text := '***';
TOF_Core.Strings.TrimChar(stringToTrim := text, trimChar := '*');
Assert.ThatBool(
	actual := text = '',
	message := "Trimming all matching characters must make the result empty"
).IsTrue();
END_METHOD

//! <summary>Borrows the concrete class name. Callers must not modify it.</summary>
{attribute 'monitoring' := 'call'}
PROPERTY ClassName : REFERENCE TO STRING
GET
ClassName REF= _ClassName;
END_GET
END_PROPERTY

//! <summary>Borrows the compiler-initialized namespace name. Callers must not modify it.</summary>
{attribute 'monitoring' := 'call'}
PROPERTY NamespaceName : REFERENCE TO STRING
GET
NamespaceName REF= CurrentNamespace.Name;
END_GET
END_PROPERTY

//! <summary>Reports the concrete instance size in bytes.</summary>
{attribute 'monitoring' := 'call'}
PROPERTY SelfSize : ULINT
GET
SelfSize := XSIZEOF(THIS^);
END_GET
END_PROPERTY

END_FUNCTION_BLOCK

// ---- Tests/Strings/String/StringSeparatorBoundsTest.TcPOU
(*
SPDX-FileCopyrightText: c 2026 Oleksandr Tiutyk <trofimich@gmail.com>
SPDX-License-Identifier: MIT
License: https://opensource.org/license/mit
*)

(*!
<summary>Checks separator length boundaries and missing borrowed sources.</summary>
<description>
Uses one task and stays at a stable address while assertions are bound to this instance.
</description>
*)

{attribute 'no_assign'}
{attribute 'no_explicit_call' := 'do not call this function block directly'}
FUNCTION_BLOCK StringSeparatorBoundsTest EXTENDS TOF_Testing.SingleCycleTest
VAR_STAT
	{attribute 'hide'}
	_ClassName : STRING := __POUNAME();
END_VAR
VAR
	_Source : STRING(82) := 'xaaaaaaaaaaaaaaaaaaaaaaaaaaaaaaaaaaaaaaaaaaaaaaaaaaaaaaaaaaaaaaaaaaaaaaaaaaaaaaaay';
	_Splitter : TOF_Core.StringSplittingEnumerator;
END_VAR

(*!
<summary>Checks separator length boundaries and missing borrowed sources.</summary>
<description>
Owns a persistent cursor and its borrowed source. The separators are bounded ASCII byte sequences.
Reset releases the current fragment before the result is reported.
</description>
*)
METHOD PROTECTED ExecuteTest
VAR
	separator : STRING(256);
	separatorUnits : POINTER TO BYTE;
	separatorLength : UINT;
	lengths : ARRAY [0..4] OF UINT := [0, 80, 81, 255, 256];
	caseLabel : WSTRING(80);
	missingSource : REFERENCE TO STRING;

	exceptionCode : __SYSTEM.ExceptionCode;
	caught : TOF_Core.IException;
	rangeException : TOF_Core.IArgumentOutOfRangeException;
	accepted : BOOL;
	i : DINT;
	j : INT;
END_VAR
// SA0175: Construct bounded ASCII separators of exact byte lengths.
{analysis -175}
separatorUnits := ADR(separator);
{analysis +175}

FOR i := 0 TO UPPER_BOUND(lengths, 1) DO
	separatorLength := lengths[i];
	caseLabel := Tc2_Utilities.WCONCAT(STR1 := "separator length ", STR2 := TO_WSTRING(separatorLength));
	FOR j := 0 TO TO_INT(separatorLength) - 1 DO
		separatorUnits[j] := BYTE#16#61;
	END_FOR

	separatorUnits[separatorLength] := TO_BYTE(TOF_Core.UnsignedInt8.MIN_VALUE);

	accepted := TOF_Core.Strings.TryCreateSplitter(sourceString := _Source, separator := separator, splitter => _Splitter);
	Assert.ThatBool(
		actual := accepted = (separatorLength = 80),
		message := Tc2_Utilities.WCONCAT(STR1 := "TryCreateSplitter at ", STR2 := caseLabel)
	).IsTrue();

	IF accepted THEN
		assertMaximumSplit(scenario := "TryCreateSplitter must use the full accepted separator");
		_Splitter.Reset();
	END_IF

	caught := 0;

	// Capture the expected argument error before inspecting the payload.
	__TRY
		_Splitter := TOF_Core.Strings.CreateSplitter(sourceString := _Source, separator := separator);
	__CATCH(exceptionCode)
		caught := TOF_Core.ExceptionManager.GetLastException(
			exceptionCode := exceptionCode,
			catchPointNamespaceName := NamespaceName,
			catchPointPOUName := __POUNAME(),
			catchPointPosition := __POSITION()
		);
	__ENDTRY

	IF separatorLength = 80 THEN
		Assert.ThatBool(actual := caught = 0, message := "CreateSplitter must accept length 80").IsTrue();

		IF caught = 0 THEN
			assertMaximumSplit(scenario := "CreateSplitter must use the full accepted separator");
			_Splitter.Reset();
		END_IF
	ELSE
		Assert.ThatBool(
			actual := __QUERYINTERFACE(caught, rangeException),
			message := Tc2_Utilities.WCONCAT(STR1 := "Expected ArgumentOutOfRangeException for ", STR2 := caseLabel)
		).IsTrue();
	END_IF
END_FOR

accepted := TOF_Core.Strings.TryCreateSplitter(
	sourceString := missingSource,
	separator := ',',
	splitter => _Splitter
);
Assert.ThatBool(
	actual := accepted,
	message := "TryCreateSplitter must return FALSE for an unbound source"
).IsFalse();
END_METHOD

(*!
<summary>Verifies that all 80 separator units are used when locating the two fragments.</summary>
<param name="scenario">Factory name included in failure messages.</param>
*)
METHOD PRIVATE assertMaximumSplit
VAR_INPUT
	scenario : WSTRING(80);
END_VAR
VAR
	entry : REFERENCE TO STRING;
	advanced : BOOL;
END_VAR
advanced := _Splitter.MoveNext();
entry REF= _Splitter.CurrentEntry;
Assert.ThatBool(
	actual := advanced AND_THEN __ISVALIDREF(entry) AND_THEN entry = 'x',
	message := scenario
).IsTrue();

advanced := _Splitter.MoveNext();
entry REF= _Splitter.CurrentEntry;
Assert.ThatBool(
	actual := advanced AND_THEN __ISVALIDREF(entry) AND_THEN entry = 'y',
	message := scenario
).IsTrue();

advanced := _Splitter.MoveNext();
Assert.ThatBool(actual := advanced, message := scenario).IsFalse();
END_METHOD

(*!
<summary>Resets the splitter and releases any active fragment before reporting.</summary>
<description>
Safe after partial initialization and after explicit cleanup in the scenario.
</description>
*)
METHOD PROTECTED AfterTest
_Splitter.Reset();
END_METHOD

//! <summary>Borrows the concrete class name. Callers must not modify it.</summary>
{attribute 'monitoring' := 'call'}
PROPERTY ClassName : REFERENCE TO STRING
GET
ClassName REF= _ClassName;
END_GET
END_PROPERTY

//! <summary>Borrows the compiler-initialized namespace name. Callers must not modify it.</summary>
{attribute 'monitoring' := 'call'}
PROPERTY NamespaceName : REFERENCE TO STRING
GET
NamespaceName REF= CurrentNamespace.Name;
END_GET
END_PROPERTY

//! <summary>Reports the concrete instance size in bytes.</summary>
{attribute 'monitoring' := 'call'}
PROPERTY SelfSize : ULINT
GET
SelfSize := XSIZEOF(THIS^);
END_GET
END_PROPERTY

END_FUNCTION_BLOCK

// ---- Tests/Strings/WideString/WideStringsTestGroup.TcPOU
(*
SPDX-FileCopyrightText: c 2026 Oleksandr Tiutyk <trofimich@gmail.com>
SPDX-License-Identifier: MIT
License: https://opensource.org/license/mit
*)

(*!
<summary>Groups wide-string formatting, editing, search and splitter contracts.</summary>
<description>
Owns the independent child instances and their fixed registration array. Use from one PLC task at a stable address.
</description>
*)

{attribute 'no_assign'}
{attribute 'no_explicit_call' := 'do not call this function block directly'}
FUNCTION_BLOCK WideStringsTestGroup EXTENDS TOF_Testing.TestGroup<11>
VAR_STAT
	{attribute 'hide'}
	_ClassName : STRING := __POUNAME();
END_VAR
VAR
	_AnyToStringFit255 : WideStringFitFormattingTest(name := "AnyToStringFit255", parent := THIS^);
	_Append : WideStringAppendTest(name := "Append", parent := THIS^);
	_AppendFit : WideStringAppendFitTest(name := "AppendFit", parent := THIS^);
	_ConcatFit255 : WideStringConcatFitTest(name := "ConcatFit255", parent := THIS^);
	_Contains : WideStringContainsTest(name := "Contains", parent := THIS^);
	_Join : WideStringJoinTest(name := "Join", parent := THIS^);
	_ReplaceInSource : WideStringReplacementTest(name := "ReplaceInSource", parent := THIS^);
	_Split : WideStringSplitTest(name := "Split", parent := THIS^);
	_Trim : WideStringTrimTest(name := "Trim", parent := THIS^);
	_SplitterSeparatorBounds : WideStringSeparatorBoundsTest(name := "SplitterSeparatorBounds", parent := THIS^);
	_AnyToStringFitLongInputs : WideStringLongFitFormattingTest(name := "AnyToStringFitLongInputs", parent := THIS^);

	_Children : ARRAY [0.._ChildCount - 1] OF TOF_Testing.ITestElement :=
	[
		_AnyToStringFit255,
		_Append,
		_AppendFit,
		_ConcatFit255,
		_Contains,
		_Join,
		_ReplaceInSource,
		_Split,
		_Trim,
		_SplitterSeparatorBounds,
		_AnyToStringFitLongInputs
	];
END_VAR

//! <summary>Borrows the fixed child array. Callers must not modify it.</summary>
{attribute 'monitoring' := 'call'}
PROPERTY Children : REFERENCE TO ARRAY [0.._ChildCount - 1] OF TOF_Testing.ITestElement
GET
Children REF= _Children;
END_GET
END_PROPERTY

//! <summary>Borrows the concrete class name. Callers must not modify it.</summary>
{attribute 'monitoring' := 'call'}
PROPERTY ClassName : REFERENCE TO STRING
GET
ClassName REF= _ClassName;
END_GET
END_PROPERTY

//! <summary>Borrows the compiler-initialized namespace name. Callers must not modify it.</summary>
{attribute 'monitoring' := 'call'}
PROPERTY NamespaceName : REFERENCE TO STRING
GET
NamespaceName REF= CurrentNamespace.Name;
END_GET
END_PROPERTY

//! <summary>Reports the concrete instance size in bytes.</summary>
{attribute 'monitoring' := 'call'}
PROPERTY SelfSize : ULINT
GET
SelfSize := XSIZEOF(THIS^);
END_GET
END_PROPERTY

END_FUNCTION_BLOCK

// ---- Tests/Strings/WideString/WideStringFitFormattingTest.TcPOU
(*
SPDX-FileCopyrightText: c 2026 Oleksandr Tiutyk <trofimich@gmail.com>
SPDX-License-Identifier: MIT
License: https://opensource.org/license/mit
*)

(*!
<summary>Checks scalar and short text formatting through the fitted ANY API.</summary>
<description>
Uses one task and stays at a stable address while assertions are bound to this instance.
</description>
*)

{attribute 'no_assign'}
{attribute 'no_explicit_call' := 'do not call this function block directly'}
FUNCTION_BLOCK WideStringFitFormattingTest EXTENDS TOF_Testing.SingleCycleTest
VAR_STAT
	{attribute 'hide'}
	_ClassName : STRING := __POUNAME();
END_VAR

(*!
<summary>Checks scalar and short text formatting through the fitted ANY API.</summary>
*)
METHOD PROTECTED ExecuteTest
VAR
	formatted : WSTRING(255);
	enabled : BOOL := TRUE;
	number : DINT := 12345;
	narrowText : STRING(50) := 'Sample string';
	wideText : WSTRING(50) := "Sample wide string";
END_VAR
formatted := TOF_Core.WideStrings.AnyToStringFit255(value := enabled);
Assert.ThatBool(
	actual := formatted = "TRUE",
	message := "AnyToStringFit255 must format BOOL"
).IsTrue();

formatted := TOF_Core.WideStrings.AnyToStringFit255(value := number);
Assert.ThatBool(
	actual := formatted = "12345",
	message := "AnyToStringFit255 must format DINT"
).IsTrue();

formatted := TOF_Core.WideStrings.AnyToStringFit255(value := narrowText);
Assert.ThatBool(
	actual := formatted = "Sample string",
	message := "AnyToStringFit255 must convert short STRING to WSTRING"
).IsTrue();

formatted := TOF_Core.WideStrings.AnyToStringFit255(value := wideText);
Assert.ThatBool(
	actual := formatted = "Sample wide string",
	message := "AnyToStringFit255 must pass short WSTRING as-is"
).IsTrue();
END_METHOD

//! <summary>Borrows the concrete class name. Callers must not modify it.</summary>
{attribute 'monitoring' := 'call'}
PROPERTY ClassName : REFERENCE TO STRING
GET
ClassName REF= _ClassName;
END_GET
END_PROPERTY

//! <summary>Borrows the compiler-initialized namespace name. Callers must not modify it.</summary>
{attribute 'monitoring' := 'call'}
PROPERTY NamespaceName : REFERENCE TO STRING
GET
NamespaceName REF= CurrentNamespace.Name;
END_GET
END_PROPERTY

//! <summary>Reports the concrete instance size in bytes.</summary>
{attribute 'monitoring' := 'call'}
PROPERTY SelfSize : ULINT
GET
SelfSize := XSIZEOF(THIS^);
END_GET
END_PROPERTY

END_FUNCTION_BLOCK

// ---- Tests/Strings/WideString/WideStringAppendTest.TcPOU
(*
SPDX-FileCopyrightText: c 2026 Oleksandr Tiutyk <trofimich@gmail.com>
SPDX-License-Identifier: MIT
License: https://opensource.org/license/mit
*)

(*!
<summary>Checks strict and Try appends, including empty fragments and capacity failure.</summary>
<description>
Uses one task and stays at a stable address while assertions are bound to this instance.
</description>
*)

{attribute 'no_assign'}
{attribute 'no_explicit_call' := 'do not call this function block directly'}
FUNCTION_BLOCK WideStringAppendTest EXTENDS TOF_Testing.SingleCycleTest
VAR_STAT
	{attribute 'hide'}
	_ClassName : STRING := __POUNAME();
END_VAR

(*!
<summary>Checks strict and Try appends, including empty fragments and capacity failure.</summary>
<description>
Both widths use small buffers to exercise the exact capacity and a failing subsequent append.
</description>
*)
METHOD PROTECTED ExecuteTest
VAR
	target : WSTRING(8);
	accepted : BOOL;
END_VAR
target := "ab";
TOF_Core.WideStrings.Append255(target, "cd", "", "efgh");
Assert.ThatBool(
	actual := target = "abcdefgh",
	message := "Append255 must skip an empty fragment and fill the target exactly"
).IsTrue();

target := "ab";
accepted := TOF_Core.WideStrings.TryAppend255(
	targetString := target,
	sourceString1 := "cd",
	sourceString2 := "",
	sourceString3 := "efgh"
);
Assert.ThatBool(
	actual := accepted AND_THEN target = "abcdefgh",
	message := "TryAppend255 must accept an exact fit"
).IsTrue();

target := "ab";
accepted := TOF_Core.WideStrings.TryAppend255(
	targetString := target,
	sourceString1 := "cd",
	sourceString2 := "ABCDE",
	sourceString3 := "!"
);
Assert.ThatBool(
	actual := accepted,
	message := "TryAppend255 must report capacity failure"
).IsFalse();
Assert.ThatBool(
	actual := Tc2_Standard.WLEFT(STR := target, SIZE := 4) = "abcd",
	message := "TryAppend255 must preserve the successfully appended prefix"
).IsTrue();

target := "ab";
TOF_Core.WideStrings.Append(targetString := target, sourceString := "cd");
TOF_Core.WideStrings.Append(targetString := target, sourceString := "");
TOF_Core.WideStrings.Append(targetString := target, sourceString := "efgh");
Assert.ThatBool(
	actual := target = "abcdefgh",
	message := "Append must preserve the target on empty input and accept the exact fit"
).IsTrue();

target := "abcdef";
accepted := TOF_Core.WideStrings.TryAppend(targetString := target, sourceString := "gh");
Assert.ThatBool(
	actual := accepted AND_THEN target = "abcdefgh",
	message := "TryAppend must accept an exact fit"
).IsTrue();

accepted := TOF_Core.WideStrings.TryAppend(targetString := target, sourceString := "i");
Assert.ThatBool(
	actual := accepted,
	message := "TryAppend must reject another character in a full target"
).IsFalse();
Assert.ThatBool(
	actual := target = "abcdefgh",
	message := "TryAppend must preserve the full target when one more character does not fit"
).IsTrue();
END_METHOD

//! <summary>Borrows the concrete class name. Callers must not modify it.</summary>
{attribute 'monitoring' := 'call'}
PROPERTY ClassName : REFERENCE TO STRING
GET
ClassName REF= _ClassName;
END_GET
END_PROPERTY

//! <summary>Borrows the compiler-initialized namespace name. Callers must not modify it.</summary>
{attribute 'monitoring' := 'call'}
PROPERTY NamespaceName : REFERENCE TO STRING
GET
NamespaceName REF= CurrentNamespace.Name;
END_GET
END_PROPERTY

//! <summary>Reports the concrete instance size in bytes.</summary>
{attribute 'monitoring' := 'call'}
PROPERTY SelfSize : ULINT
GET
SelfSize := XSIZEOF(THIS^);
END_GET
END_PROPERTY

END_FUNCTION_BLOCK

// ---- Tests/Strings/WideString/WideStringAppendFitTest.TcPOU
(*
SPDX-FileCopyrightText: c 2026 Oleksandr Tiutyk <trofimich@gmail.com>
SPDX-License-Identifier: MIT
License: https://opensource.org/license/mit
*)

(*!
<summary>Checks fitted appends at exact capacity and on truncation.</summary>
<description>
Uses one task and stays at a stable address while assertions are bound to this instance.
</description>
*)

{attribute 'no_assign'}
{attribute 'no_explicit_call' := 'do not call this function block directly'}
FUNCTION_BLOCK WideStringAppendFitTest EXTENDS TOF_Testing.SingleCycleTest
VAR_STAT
	{attribute 'hide'}
	_ClassName : STRING := __POUNAME();
END_VAR

(*!
<summary>Checks fitted appends at exact capacity and on truncation.</summary>
*)
METHOD PROTECTED ExecuteTest
VAR
	oneCharacter : WSTRING(1);
	twoCharacters : WSTRING(2);
	target : WSTRING(10);
	longFragment : WSTRING(30) := "01234567890123456789";
	accepted : BOOL;
END_VAR
// Fits within capacity
target := "12345";
TOF_Core.WideStrings.AppendFit(targetString := target, sourceString := "67");
Assert.ThatBool(
	actual := target = "1234567",
	message := "AppendFit must append normally when it fits"
).IsTrue();

// Exact fit: fills capacity without ellipsis
target := "12345";
TOF_Core.WideStrings.AppendFit(targetString := target, sourceString := "67890");
Assert.ThatBool(
	actual := target = "1234567890",
	message := "AppendFit must fit exactly without ellipsis"
).IsTrue();

// Overflow by one code unit uses U+2026.
target := "12345";
TOF_Core.WideStrings.AppendFit(targetString := target, sourceString := "678901");
Assert.ThatBool(
	actual := target = "123456789$2026",
	message := "AppendFit must truncate and append ellipsis on 1 char overflow"
).IsTrue();

// A larger overflow still uses one U+2026 code unit.
target := "12345";
TOF_Core.WideStrings.AppendFit(targetString := target, sourceString := longFragment);
Assert.ThatBool(
	actual := target = "123450123$2026",
	message := "AppendFit must truncate and append ellipsis on large overflow"
).IsTrue();

// Empty source: target remains unchanged
target := "12345";
TOF_Core.WideStrings.AppendFit(targetString := target, sourceString := "");
Assert.ThatBool(
	actual := target = "12345",
	message := "AppendFit must leave target unchanged for empty source"
).IsTrue();

// Appending to empty target
target := "";
TOF_Core.WideStrings.AppendFit(targetString := target, sourceString := longFragment);
Assert.ThatBool(
	actual := target = "012345678$2026",
	message := "AppendFit to empty target must truncate and append ellipsis"
).IsTrue();

// TryAppendFit normal fit
target := "123";
accepted := TOF_Core.WideStrings.TryAppendFit(targetString := target, sourceString := "45");
Assert.ThatBool(
	actual := accepted,
	message := "TryAppendFit must return TRUE on normal fit"
).IsTrue();
Assert.ThatBool(
	actual := target = "12345",
	message := "TryAppendFit must append text"
).IsTrue();

// TryAppendFit overflow
target := "12345";
accepted := TOF_Core.WideStrings.TryAppendFit(targetString := target, sourceString := longFragment);
Assert.ThatBool(
	actual := accepted,
	message := "TryAppendFit must return TRUE on overflow"
).IsTrue();
Assert.ThatBool(
	actual := target = "123450123$2026",
	message := "TryAppendFit must truncate and append ellipsis"
).IsTrue();

// AppendFit255 multiple arguments and literals
target := "12";
TOF_Core.WideStrings.AppendFit255(target, "3", "4", "5");
Assert.ThatBool(
	actual := target = "12345",
	message := "AppendFit255 must append multiple fragments"
).IsTrue();

// AppendFit255 overflow truncation
target := "12";
TOF_Core.WideStrings.AppendFit255(target, "345", "678", "9012");
Assert.ThatBool(
	actual := target = "123456789$2026",
	message := "AppendFit255 must truncate and append ellipsis on overflow"
).IsTrue();

// TryAppendFit255 normal fit
target := "12";
accepted := TOF_Core.WideStrings.TryAppendFit255(
	targetString := target,
	sourceString1 := "3",
	sourceString2 := "4",
	sourceString3 := "5"
);
Assert.ThatBool(
	actual := accepted,
	message := "TryAppendFit255 must return TRUE on normal fit"
).IsTrue();
Assert.ThatBool(
	actual := target = "12345",
	message := "TryAppendFit255 must append multiple fragments"
).IsTrue();

// TryAppendFit255 overflow
target := "12";
accepted := TOF_Core.WideStrings.TryAppendFit255(
	targetString := target,
	sourceString1 := "345",
	sourceString2 := "678",
	sourceString3 := "9012"
);
Assert.ThatBool(
	actual := accepted,
	message := "TryAppendFit255 must return TRUE on overflow"
).IsTrue();
Assert.ThatBool(
	actual := target = "123456789$2026",
	message := "TryAppendFit255 must truncate and append ellipsis on overflow"
).IsTrue();

accepted := TOF_Core.WideStrings.TryAppendFit(targetString := oneCharacter, sourceString := longFragment);
Assert.ThatBool(
	actual := accepted,
	message := "Truncation must succeed in a one-character buffer"
).IsTrue();
Assert.ThatBool(
	actual := oneCharacter = "$2026",
	message := "One-character truncation marker"
).IsTrue();

accepted := TOF_Core.WideStrings.TryAppendFit255(targetString := twoCharacters, sourceString1 := longFragment);
Assert.ThatBool(
	actual := accepted,
	message := "Truncation must succeed in a two-character buffer"
).IsTrue();
Assert.ThatBool(
	actual := twoCharacters = "0$2026",
	message := "Two-character truncation marker"
).IsTrue();
END_METHOD

//! <summary>Borrows the concrete class name. Callers must not modify it.</summary>
{attribute 'monitoring' := 'call'}
PROPERTY ClassName : REFERENCE TO STRING
GET
ClassName REF= _ClassName;
END_GET
END_PROPERTY

//! <summary>Borrows the compiler-initialized namespace name. Callers must not modify it.</summary>
{attribute 'monitoring' := 'call'}
PROPERTY NamespaceName : REFERENCE TO STRING
GET
NamespaceName REF= CurrentNamespace.Name;
END_GET
END_PROPERTY

//! <summary>Reports the concrete instance size in bytes.</summary>
{attribute 'monitoring' := 'call'}
PROPERTY SelfSize : ULINT
GET
SelfSize := XSIZEOF(THIS^);
END_GET
END_PROPERTY

END_FUNCTION_BLOCK

// ---- Tests/Strings/WideString/WideStringConcatFitTest.TcPOU
(*
SPDX-FileCopyrightText: c 2026 Oleksandr Tiutyk <trofimich@gmail.com>
SPDX-License-Identifier: MIT
License: https://opensource.org/license/mit
*)

(*!
<summary>Checks fitted concatenation, including the 255-character boundary.</summary>
<description>
Uses one task and stays at a stable address while assertions are bound to this instance.
</description>
*)

{attribute 'no_assign'}
{attribute 'no_explicit_call' := 'do not call this function block directly'}
FUNCTION_BLOCK WideStringConcatFitTest EXTENDS TOF_Testing.SingleCycleTest
VAR_STAT
	{attribute 'hide'}
	_ClassName : STRING := __POUNAME();
END_VAR

(*!
<summary>Checks fitted concatenation, including the 255-character boundary.</summary>
<description>
Distinct fragments reveal the first discarded character and any changes in fragment order.
</description>
*)
METHOD PROTECTED ExecuteTest
VAR
	text : WSTRING(255);
	first : WSTRING(100) := "aaaaaaaaaaaaaaaaaaaaaaaaaaaaaaaaaaaaaaaaaaaaaaaaaaaaaaaaaaaaaaaaaaaaaaaaaaaaaaaaaaaaaaaaaaaaaaaaaaaa";
	second : WSTRING(100) := "bbbbbbbbbbbbbbbbbbbbbbbbbbbbbbbbbbbbbbbbbbbbbbbbbbbbbbbbbbbbbbbbbbbbbbbbbbbbbbbbbbbbbbbbbbbbbbbbbbbb";
	third : WSTRING(100) := "cccccccccccccccccccccccccccccccccccccccccccccccccccccccccccccccccccccccccccccccccccccccccccccccccccc";
	expectedPrefix : WSTRING(255);
END_VAR
text := TOF_Core.WideStrings.ConcatFit255("Hello, ", "World!");
Assert.ThatBool(
	actual := text = "Hello, World!",
	message := "ConcatFit255 must preserve an ordinary fit"
).IsTrue();

text := TOF_Core.WideStrings.ConcatFit255("Part1", "", "Part2", "", "Part3");
Assert.ThatBool(
	actual := text = "Part1Part2Part3",
	message := "ConcatFit255 must skip empty fragments without stopping"
).IsTrue();

text := TOF_Core.WideStrings.ConcatFit255(first, second, third);
Assert.ThatInt(
	actual := Tc2_Standard.WLEN(STR := text),
	message := "ConcatFit255 must fill the 255-character result"
).ToBe(expected := 255);
expectedPrefix := Tc2_Standard.WCONCAT(STR1 := first, STR2 := second);
expectedPrefix := Tc2_Standard.WCONCAT(
	STR1 := expectedPrefix,
	STR2 := Tc2_Standard.WLEFT(STR := third, SIZE := 54)
);
Assert.ThatBool(
	actual := Tc2_Standard.WLEFT(STR := text, SIZE := 254) = expectedPrefix,
	message := "Truncation must preserve the prefix across all three fragments"
).IsTrue();
Assert.ThatBool(
	actual := Tc2_Standard.WRIGHT(STR := text, SIZE := 1) = "$2026",
	message := "Truncation must use the exact encoding-specific ellipsis"
).IsTrue();
END_METHOD

//! <summary>Borrows the concrete class name. Callers must not modify it.</summary>
{attribute 'monitoring' := 'call'}
PROPERTY ClassName : REFERENCE TO STRING
GET
ClassName REF= _ClassName;
END_GET
END_PROPERTY

//! <summary>Borrows the compiler-initialized namespace name. Callers must not modify it.</summary>
{attribute 'monitoring' := 'call'}
PROPERTY NamespaceName : REFERENCE TO STRING
GET
NamespaceName REF= CurrentNamespace.Name;
END_GET
END_PROPERTY

//! <summary>Reports the concrete instance size in bytes.</summary>
{attribute 'monitoring' := 'call'}
PROPERTY SelfSize : ULINT
GET
SelfSize := XSIZEOF(THIS^);
END_GET
END_PROPERTY

END_FUNCTION_BLOCK

// ---- Tests/Strings/WideString/WideStringContainsTest.TcPOU
(*
SPDX-FileCopyrightText: c 2026 Oleksandr Tiutyk <trofimich@gmail.com>
SPDX-License-Identifier: MIT
License: https://opensource.org/license/mit
*)

(*!
<summary>Checks exact, case-sensitive substring matching and empty inputs.</summary>
<description>
Uses one task and stays at a stable address while assertions are bound to this instance.
</description>
*)

{attribute 'no_assign'}
{attribute 'no_explicit_call' := 'do not call this function block directly'}
FUNCTION_BLOCK WideStringContainsTest EXTENDS TOF_Testing.SingleCycleTest
VAR_STAT
	{attribute 'hide'}
	_ClassName : STRING := __POUNAME();
END_VAR

(*!
<summary>Checks exact, case-sensitive substring matching and empty inputs.</summary>
*)
METHOD PROTECTED ExecuteTest
VAR
	containsResult : BOOL;
END_VAR
containsResult := TOF_Core.WideStrings.Contains(stringToSearchIn := "Hello, world!", stringToFind := "Hello");
Assert.ThatBool(
	actual := containsResult,
	message := "Contains must return TRUE for prefix substring"
).IsTrue();

containsResult := TOF_Core.WideStrings.Contains(stringToSearchIn := "Hello, world!", stringToFind := "world");
Assert.ThatBool(
	actual := containsResult,
	message := "Contains must return TRUE for middle substring"
).IsTrue();

containsResult := TOF_Core.WideStrings.Contains(stringToSearchIn := "Hello, world!", stringToFind := "!");
Assert.ThatBool(
	actual := containsResult,
	message := "Contains must return TRUE for suffix substring"
).IsTrue();

containsResult := TOF_Core.WideStrings.Contains(stringToSearchIn := "Hello, world!", stringToFind := "Hello, world!");
Assert.ThatBool(
	actual := containsResult,
	message := "Contains must return TRUE for identical string"
).IsTrue();

containsResult := TOF_Core.WideStrings.Contains(stringToSearchIn := "Hello, world!", stringToFind := "");
Assert.ThatBool(
	actual := containsResult,
	message := "Contains must return TRUE for empty substring in non-empty string"
).IsTrue();

containsResult := TOF_Core.WideStrings.Contains(stringToSearchIn := "", stringToFind := "");
Assert.ThatBool(
	actual := containsResult,
	message := "Contains must return TRUE for empty substring in empty string"
).IsTrue();

containsResult := TOF_Core.WideStrings.Contains(stringToSearchIn := "", stringToFind := "a");
Assert.ThatBool(
	actual := containsResult,
	message := "Contains must return FALSE for non-empty substring in empty string"
).IsFalse();

containsResult := TOF_Core.WideStrings.Contains(stringToSearchIn := "Hello, world!", stringToFind := "xyz");
Assert.ThatBool(
	actual := containsResult,
	message := "Contains must return FALSE when substring is absent"
).IsFalse();

containsResult := TOF_Core.WideStrings.Contains(stringToSearchIn := "Hello, world!", stringToFind := "hello");
Assert.ThatBool(
	actual := containsResult,
	message := "Contains must be case-sensitive"
).IsFalse();

containsResult := TOF_Core.WideStrings.Contains(stringToSearchIn := "abc", stringToFind := "abcdef");
Assert.ThatBool(
	actual := containsResult,
	message := "Contains must return FALSE when substring is longer than source"
).IsFalse();

containsResult := TOF_Core.WideStrings.Contains(stringToSearchIn := "aaab", stringToFind := "aab");
Assert.ThatBool(
	actual := containsResult,
	message := "Contains must restart after a partially matching prefix"
).IsTrue();
END_METHOD

//! <summary>Borrows the concrete class name. Callers must not modify it.</summary>
{attribute 'monitoring' := 'call'}
PROPERTY ClassName : REFERENCE TO STRING
GET
ClassName REF= _ClassName;
END_GET
END_PROPERTY

//! <summary>Borrows the compiler-initialized namespace name. Callers must not modify it.</summary>
{attribute 'monitoring' := 'call'}
PROPERTY NamespaceName : REFERENCE TO STRING
GET
NamespaceName REF= CurrentNamespace.Name;
END_GET
END_PROPERTY

//! <summary>Reports the concrete instance size in bytes.</summary>
{attribute 'monitoring' := 'call'}
PROPERTY SelfSize : ULINT
GET
SelfSize := XSIZEOF(THIS^);
END_GET
END_PROPERTY

END_FUNCTION_BLOCK

// ---- Tests/Strings/WideString/WideStringJoinTest.TcPOU
(*
SPDX-FileCopyrightText: c 2026 Oleksandr Tiutyk <trofimich@gmail.com>
SPDX-License-Identifier: MIT
License: https://opensource.org/license/mit
*)

(*!
<summary>Checks full and windowed joining and cursor reuse after insufficient capacity.</summary>
<description>
Uses one task and stays at a stable address while assertions are bound to this instance.
</description>
*)

{attribute 'no_assign'}
{attribute 'no_explicit_call' := 'do not call this function block directly'}
FUNCTION_BLOCK WideStringJoinTest EXTENDS TOF_Testing.SingleCycleTest
VAR_STAT
	{attribute 'hide'}
	_ClassName : STRING := __POUNAME();
END_VAR
VAR
	_Source : WSTRING := "123 , , 456, 789 ,0";
	_Splitter : TOF_Core.WideStringSplittingEnumerator;
END_VAR

(*!
<summary>Checks full and windowed joining and cursor reuse after insufficient capacity.</summary>
<description>
Owns a persistent cursor and its borrowed source. Reset releases the current fragment before the result is reported.
</description>
*)
METHOD PROTECTED ExecuteTest
VAR
	separator : WSTRING := ",";
	joined : WSTRING := "old target";
	shortTarget : WSTRING(2);
	accepted : BOOL;
END_VAR
_Splitter := TOF_Core.WideStrings.CreateSplitter(sourceString := _Source, separator := separator);
TOF_Core.WideStrings.Join(targetString := joined, separator := separator, sourceEnumerator := _Splitter);
Assert.ThatBool(
	actual := joined = _Source,
	message := "Unrestricted Join must reconstruct all fragments including their whitespace"
).IsTrue();

_Splitter.Reset();
_Splitter := TOF_Core.WideStrings.CreateSplitter(
	sourceString := _Source,
	separator := separator,
	maxCount := 3,
	trimEntries := TRUE,
	removeEmptyEntries := TRUE
);
TOF_Core.WideStrings.Join(
	targetString := joined,
	separator := separator,
	sourceEnumerator := _Splitter,
	startIndex := 1,
	count := 2
);
Assert.ThatBool(
	actual := joined = "456,789",
	message := "The requested window must contain fragments 1 and 2"
).IsTrue();

_Splitter.Reset();
accepted := TOF_Core.WideStrings.TryJoin(targetString := shortTarget, separator := separator, sourceEnumerator := _Splitter);
Assert.ThatBool(
	actual := accepted,
	message := "TryJoin must reject a target too small for the first fragment"
).IsFalse();

_Splitter.Reset();
accepted := TOF_Core.WideStrings.TryJoin(
	targetString := joined,
	separator := separator,
	sourceEnumerator := _Splitter,
	count := 1
);
Assert.ThatBool(
	actual := accepted AND_THEN joined = "123",
	message := "After Reset, TryJoin must restart and replace the old target text"
).IsTrue();
END_METHOD

(*!
<summary>Resets the splitter and releases any active fragment before reporting.</summary>
<description>
Safe after partial initialization and after explicit cleanup in the scenario.
</description>
*)
METHOD PROTECTED AfterTest
_Splitter.Reset();
END_METHOD

//! <summary>Borrows the concrete class name. Callers must not modify it.</summary>
{attribute 'monitoring' := 'call'}
PROPERTY ClassName : REFERENCE TO STRING
GET
ClassName REF= _ClassName;
END_GET
END_PROPERTY

//! <summary>Borrows the compiler-initialized namespace name. Callers must not modify it.</summary>
{attribute 'monitoring' := 'call'}
PROPERTY NamespaceName : REFERENCE TO STRING
GET
NamespaceName REF= CurrentNamespace.Name;
END_GET
END_PROPERTY

//! <summary>Reports the concrete instance size in bytes.</summary>
{attribute 'monitoring' := 'call'}
PROPERTY SelfSize : ULINT
GET
SelfSize := XSIZEOF(THIS^);
END_GET
END_PROPERTY

END_FUNCTION_BLOCK

// ---- Tests/Strings/WideString/WideStringReplacementTest.TcPOU
(*
SPDX-FileCopyrightText: c 2026 Oleksandr Tiutyk <trofimich@gmail.com>
SPDX-License-Identifier: MIT
License: https://opensource.org/license/mit
*)

(*!
<summary>Checks in-place replacements, counts, limits and partial capacity failure.</summary>
<description>
Uses one task and stays at a stable address while assertions are bound to this instance.
</description>
*)

{attribute 'no_assign'}
{attribute 'no_explicit_call' := 'do not call this function block directly'}
FUNCTION_BLOCK WideStringReplacementTest EXTENDS TOF_Testing.SingleCycleTest
VAR_STAT
	{attribute 'hide'}
	_ClassName : STRING := __POUNAME();
END_VAR

(*!
<summary>Checks in-place replacements, counts, limits and partial capacity failure.</summary>
<description>
Uses caller-owned buffers with known capacities. A failed next replacement must leave earlier matches applied.
</description>
*)
METHOD PROTECTED ExecuteTest
VAR
	text : WSTRING(18);
	
	replacementCount : UINT;
	result : BOOL;
END_VAR
text := "abcd_abcd_abcd";
TOF_Core.WideStrings.ReplaceInSource(
	sourceString := text,
	oldSubstring := "bc",
	newSubstring := "0",
	replacementCount => replacementCount
);
Assert.ThatBool(
	actual := text = "a0d_a0d_a0d",
	message := "Shrink must produce the expected text"
).IsTrue();
Assert.ThatUInt(
	actual := replacementCount,
	message := "Shrink must produce the expected count"
).ToBe(expected := 3);

text := "abcd_abcd_abcd";
TOF_Core.WideStrings.ReplaceInSource(
	sourceString := text,
	oldSubstring := "bc",
	newSubstring := "123",
	replacementCount => replacementCount
);
Assert.ThatBool(
	actual := text = "a123d_a123d_a123d",
	message := "Grow must produce the expected text"
).IsTrue();
Assert.ThatUInt(
	actual := replacementCount,
	message := "Grow must produce the expected count"
).ToBe(expected := 3);

text := "abcd_abcd_abcd";
result := TOF_Core.WideStrings.TryReplaceInSource(
	sourceString := text,
	oldSubstring := "bc",
	newSubstring := "0",
	replacementCount => replacementCount
);
Assert.ThatBool(
	actual := result,
	message := "Try shrink must produce the expected status"
).IsTrue();
Assert.ThatBool(
	actual := text = "a0d_a0d_a0d",
	message := "Try shrink must produce the expected text"
).IsTrue();
Assert.ThatUInt(
	actual := replacementCount,
	message := "Try shrink must produce the expected count"
).ToBe(expected := 3);

text := "abcd_abcd_abcd";
result := TOF_Core.WideStrings.TryReplaceInSource(
	sourceString := text,
	oldSubstring := "bc",
	newSubstring := "123",
	maxReplacements := 1,
	skipReplacements := 1,
	replacementCount => replacementCount
);
Assert.ThatBool(
	actual := result,
	message := "Try skip and limit must produce the expected status"
).IsTrue();
Assert.ThatBool(
	actual := text = "abcd_a123d_abcd",
	message := "Try skip and limit must produce the expected text"
).IsTrue();
Assert.ThatUInt(
	actual := replacementCount,
	message := "Try skip and limit must produce the expected count"
).ToBe(expected := 1);

text := "abcd_abcd_abcd";
result := TOF_Core.WideStrings.TryReplaceInSource(
	sourceString := text,
	oldSubstring := "bc",
	newSubstring := "1234",
	replacementCount => replacementCount
);
Assert.ThatBool(
	actual := result,
	message := "Growth must report failure when the next replacement exceeds capacity"
).IsFalse();
Assert.ThatBool(
	actual := text = "a1234d_a1234d_abcd",
	message := "Capacity failure must preserve both completed replacements"
).IsTrue();
Assert.ThatUInt(
	actual := replacementCount,
	message := "Capacity failure must report both completed replacements"
).ToBe(expected := UINT#2);

text := "abcd_abcd";
result := TOF_Core.WideStrings.TryReplaceInSource(
	sourceString := text,
	oldSubstring := "",
	newSubstring := "ignore",
	replacementCount => replacementCount
);
Assert.ThatBool(
	actual := result AND_THEN text = "abcd_abcd" AND_THEN replacementCount = 0,
	message := "An empty search must succeed without modifying text or reporting replacements"
).IsTrue();

result := TOF_Core.WideStrings.TryReplaceInSource(
	sourceString := text,
	oldSubstring := "bc",
	newSubstring := "",
	replacementCount => replacementCount
);
Assert.ThatBool(
	actual := result AND_THEN text = "ad_ad" AND_THEN replacementCount = 2,
	message := "An empty replacement must delete both matching substrings"
).IsTrue();
END_METHOD

//! <summary>Borrows the concrete class name. Callers must not modify it.</summary>
{attribute 'monitoring' := 'call'}
PROPERTY ClassName : REFERENCE TO STRING
GET
ClassName REF= _ClassName;
END_GET
END_PROPERTY

//! <summary>Borrows the compiler-initialized namespace name. Callers must not modify it.</summary>
{attribute 'monitoring' := 'call'}
PROPERTY NamespaceName : REFERENCE TO STRING
GET
NamespaceName REF= CurrentNamespace.Name;
END_GET
END_PROPERTY

//! <summary>Reports the concrete instance size in bytes.</summary>
{attribute 'monitoring' := 'call'}
PROPERTY SelfSize : ULINT
GET
SelfSize := XSIZEOF(THIS^);
END_GET
END_PROPERTY

END_FUNCTION_BLOCK

// ---- Tests/Strings/WideString/WideStringSplitTest.TcPOU
(*
SPDX-FileCopyrightText: c 2026 Oleksandr Tiutyk <trofimich@gmail.com>
SPDX-License-Identifier: MIT
License: https://opensource.org/license/mit
*)

(*!
<summary>Checks split fragments, end-of-iteration behavior and cursor restart.</summary>
<description>
Uses one task and stays at a stable address while assertions are bound to this instance.
</description>
*)

{attribute 'no_assign'}
{attribute 'no_explicit_call' := 'do not call this function block directly'}
FUNCTION_BLOCK WideStringSplitTest EXTENDS TOF_Testing.SingleCycleTest
VAR_STAT
	{attribute 'hide'}
	_ClassName : STRING := __POUNAME();
END_VAR
VAR
	_Source : WSTRING := "123 , 456, 789 ,,0,";
	_Splitter : TOF_Core.WideStringSplittingEnumerator;
END_VAR

(*!
<summary>Checks split fragments, end-of-iteration behavior and cursor restart.</summary>
<description>
Owns a persistent cursor and its borrowed source. Reset releases the current fragment before the result is reported.
</description>
*)
METHOD PROTECTED ExecuteTest
VAR
	separator : WSTRING := ",";
	allFragments : ARRAY [0..5] OF WSTRING := ["123 ", " 456", " 789 ", "", "0", ""];
	selectedFragments : ARRAY [0..2] OF WSTRING := ["123", "456", "789"];
	entry : REFERENCE TO WSTRING;
	advanced : BOOL;
END_VAR
_Splitter := TOF_Core.WideStrings.CreateSplitter(sourceString := _Source, separator := separator);
assertFragments(expected := allFragments, scenario := "Unrestricted split");

_Splitter.Reset();
_Splitter := TOF_Core.WideStrings.CreateSplitter(
	sourceString := _Source,
	separator := separator,
	maxCount := 3,
	trimEntries := TRUE,
	removeEmptyEntries := TRUE
);
assertFragments(expected := selectedFragments, scenario := "Trimmed split limited to three");

_Splitter.Reset();
entry REF= _Splitter.CurrentEntry;
Assert.ThatBool(
	actual := __ISVALIDREF(entry),
	message := "Reset must leave CurrentEntry invalid until the next successful move"
).IsFalse();

advanced := _Splitter.MoveNext();
entry REF= _Splitter.CurrentEntry;
Assert.ThatBool(
	actual := advanced AND_THEN __ISVALIDREF(entry) AND_THEN entry = "123",
	message := "After Reset the first trimmed fragment must be available again"
).IsTrue();
END_METHOD

(*!
<summary>Checks the requested finite sequence and detects trailing fragments or a stale current reference.</summary>
<param name="expected">Expected fragments in order.</param>
<param name="scenario">Cursor configuration included in failure messages.</param>
*)
METHOD PRIVATE assertFragments
VAR_IN_OUT CONSTANT
	expected : ARRAY [*] OF WSTRING;
END_VAR
VAR_INPUT
	scenario : WSTRING(80);
END_VAR
VAR
	entry : REFERENCE TO WSTRING;
	i : DINT;
	advanced : BOOL;
	fragmentLabel : WSTRING(255);
END_VAR
FOR i := LOWER_BOUND(expected, 1) TO UPPER_BOUND(expected, 1) DO
	fragmentLabel := Tc2_Utilities.WCONCAT(STR1 := scenario, STR2 := " fragment ");
	fragmentLabel := Tc2_Utilities.WCONCAT(STR1 := fragmentLabel, STR2 := TO_WSTRING(i));
	advanced := _Splitter.MoveNext();
	Assert.ThatBool(actual := advanced, message := fragmentLabel).IsTrue();

	IF NOT advanced THEN
		RETURN;
	END_IF

	entry REF= _Splitter.CurrentEntry;
	Assert.ThatBool(actual := __ISVALIDREF(entry) AND_THEN entry = expected[i], message := fragmentLabel).IsTrue();
END_FOR

advanced := _Splitter.MoveNext();
Assert.ThatBool(
	actual := advanced,
	message := Tc2_Utilities.WCONCAT(STR1 := "Unexpected extra fragment in ", STR2 := scenario)
).IsFalse();

IF advanced THEN
	RETURN;
END_IF

entry REF= _Splitter.CurrentEntry;
Assert.ThatBool(actual := __ISVALIDREF(entry), message := "End of iteration must invalidate CurrentEntry").IsFalse();
advanced := _Splitter.MoveNext();
Assert.ThatBool(actual := advanced, message := "An exhausted splitter must stay exhausted").IsFalse();
END_METHOD

(*!
<summary>Resets the splitter and releases any active fragment before reporting.</summary>
<description>
Safe after partial initialization and after explicit cleanup in the scenario.
</description>
*)
METHOD PROTECTED AfterTest
_Splitter.Reset();
END_METHOD

//! <summary>Borrows the concrete class name. Callers must not modify it.</summary>
{attribute 'monitoring' := 'call'}
PROPERTY ClassName : REFERENCE TO STRING
GET
ClassName REF= _ClassName;
END_GET
END_PROPERTY

//! <summary>Borrows the compiler-initialized namespace name. Callers must not modify it.</summary>
{attribute 'monitoring' := 'call'}
PROPERTY NamespaceName : REFERENCE TO STRING
GET
NamespaceName REF= CurrentNamespace.Name;
END_GET
END_PROPERTY

//! <summary>Reports the concrete instance size in bytes.</summary>
{attribute 'monitoring' := 'call'}
PROPERTY SelfSize : ULINT
GET
SelfSize := XSIZEOF(THIS^);
END_GET
END_PROPERTY

END_FUNCTION_BLOCK

// ---- Tests/Strings/WideString/WideStringTrimTest.TcPOU
(*
SPDX-FileCopyrightText: c 2026 Oleksandr Tiutyk <trofimich@gmail.com>
SPDX-License-Identifier: MIT
License: https://opensource.org/license/mit
*)

(*!
<summary>Checks trimming direction, custom characters and complete removal.</summary>
<description>
Uses one task and stays at a stable address while assertions are bound to this instance.
</description>
*)

{attribute 'no_assign'}
{attribute 'no_explicit_call' := 'do not call this function block directly'}
FUNCTION_BLOCK WideStringTrimTest EXTENDS TOF_Testing.SingleCycleTest
VAR_STAT
	{attribute 'hide'}
	_ClassName : STRING := __POUNAME();
END_VAR

(*!
<summary>Checks trimming direction, custom characters and complete removal.</summary>
*)
METHOD PROTECTED ExecuteTest
VAR
	text : WSTRING;
END_VAR
text := "  123   ";
TOF_Core.WideStrings.TrimChar(stringToTrim := text, trimMode := TOF_Core.TRIM_MODE.LEFT_AND_RIGHT);
Assert.ThatBool(
	actual := text = "123",
	message := "TrimChar must apply LEFT_AND_RIGHT exactly"
).IsTrue();

text := "  123   ";
TOF_Core.WideStrings.TrimChar(stringToTrim := text, trimMode := TOF_Core.TRIM_MODE.LEFT);
Assert.ThatBool(
	actual := text = "123   ",
	message := "TrimChar must apply LEFT exactly"
).IsTrue();

text := "  123   ";
TOF_Core.WideStrings.TrimChar(stringToTrim := text, trimMode := TOF_Core.TRIM_MODE.RIGHT);
Assert.ThatBool(
	actual := text = "  123",
	message := "TrimChar must apply RIGHT exactly"
).IsTrue();

text := "**a*b**";
TOF_Core.WideStrings.TrimChar(stringToTrim := text, trimMode := TOF_Core.TRIM_MODE.LEFT_AND_RIGHT, trimChar := "*");
Assert.ThatBool(
	actual := text = "a*b",
	message := "Trimming a custom character must preserve an internal match"
).IsTrue();

text := "***";
TOF_Core.WideStrings.TrimChar(stringToTrim := text, trimChar := "*");
Assert.ThatBool(
	actual := text = "",
	message := "Trimming all matching characters must make the result empty"
).IsTrue();
END_METHOD

//! <summary>Borrows the concrete class name. Callers must not modify it.</summary>
{attribute 'monitoring' := 'call'}
PROPERTY ClassName : REFERENCE TO STRING
GET
ClassName REF= _ClassName;
END_GET
END_PROPERTY

//! <summary>Borrows the compiler-initialized namespace name. Callers must not modify it.</summary>
{attribute 'monitoring' := 'call'}
PROPERTY NamespaceName : REFERENCE TO STRING
GET
NamespaceName REF= CurrentNamespace.Name;
END_GET
END_PROPERTY

//! <summary>Reports the concrete instance size in bytes.</summary>
{attribute 'monitoring' := 'call'}
PROPERTY SelfSize : ULINT
GET
SelfSize := XSIZEOF(THIS^);
END_GET
END_PROPERTY

END_FUNCTION_BLOCK

// ---- Tests/Strings/WideString/WideStringSeparatorBoundsTest.TcPOU
(*
SPDX-FileCopyrightText: c 2026 Oleksandr Tiutyk <trofimich@gmail.com>
SPDX-License-Identifier: MIT
License: https://opensource.org/license/mit
*)

(*!
<summary>Checks separator length boundaries and missing borrowed sources.</summary>
<description>
Uses one task and stays at a stable address while assertions are bound to this instance.
</description>
*)

{attribute 'no_assign'}
{attribute 'no_explicit_call' := 'do not call this function block directly'}
FUNCTION_BLOCK WideStringSeparatorBoundsTest EXTENDS TOF_Testing.SingleCycleTest
VAR_STAT
	{attribute 'hide'}
	_ClassName : STRING := __POUNAME();
END_VAR
VAR
	_Source : WSTRING(82) := "xaaaaaaaaaaaaaaaaaaaaaaaaaaaaaaaaaaaaaaaaaaaaaaaaaaaaaaaaaaaaaaaaaaaaaaaaaaaaaaaay";
	_Splitter : TOF_Core.WideStringSplittingEnumerator;
END_VAR

(*!
<summary>Checks separator length boundaries and missing borrowed sources.</summary>
<description>
Owns a persistent cursor and its borrowed source. Reset releases the current fragment before the result is reported.
</description>
*)
METHOD PROTECTED ExecuteTest
VAR
	separator : WSTRING(256);
	separatorUnits : POINTER TO WORD;
	separatorLength : UINT;
	lengths : ARRAY [0..4] OF UINT := [0, 80, 81, 255, 256];
	caseLabel : WSTRING(80);
	missingSource : REFERENCE TO WSTRING;

	exceptionCode : __SYSTEM.ExceptionCode;
	caught : TOF_Core.IException;
	rangeException : TOF_Core.IArgumentOutOfRangeException;
	accepted : BOOL;
	i : DINT;
	j : INT;
END_VAR
separatorUnits := ADR(separator);

FOR i := 0 TO UPPER_BOUND(lengths, 1) DO
	separatorLength := lengths[i];
	caseLabel := Tc2_Utilities.WCONCAT(STR1 := "separator length ", STR2 := TO_WSTRING(separatorLength));

	FOR j := 0 TO TO_INT(separatorLength) - 1 DO
		separatorUnits[j] := WORD#16#0061;
	END_FOR

	separatorUnits[separatorLength] := TO_WORD(TOF_Core.UnsignedInt16.MIN_VALUE);

	accepted := TOF_Core.WideStrings.TryCreateSplitter(sourceString := _Source, separator := separator, splitter => _Splitter);
	Assert.ThatBool(
		actual := accepted = (separatorLength = 80),
		message := Tc2_Utilities.WCONCAT(STR1 := "TryCreateSplitter at ", STR2 := caseLabel)
	).IsTrue();

	IF accepted THEN
		assertMaximumSplit(scenario := "TryCreateSplitter must use the full accepted separator");
		_Splitter.Reset();
	END_IF

	caught := 0;

	// Capture the expected argument error before inspecting the payload.
	__TRY
		_Splitter := TOF_Core.WideStrings.CreateSplitter(sourceString := _Source, separator := separator);
	__CATCH(exceptionCode)
		caught := TOF_Core.ExceptionManager.GetLastException(
			exceptionCode := exceptionCode,
			catchPointNamespaceName := NamespaceName,
			catchPointPOUName := __POUNAME(),
			catchPointPosition := __POSITION()
		);
	__ENDTRY

	IF separatorLength = 80 THEN
		Assert.ThatBool(actual := caught = 0, message := "CreateSplitter must accept length 80").IsTrue();

		IF caught = 0 THEN
			assertMaximumSplit(scenario := "CreateSplitter must use the full accepted separator");
			_Splitter.Reset();
		END_IF
	ELSE
		Assert.ThatBool(
			actual := __QUERYINTERFACE(caught, rangeException),
			message := Tc2_Utilities.WCONCAT(STR1 := "Expected ArgumentOutOfRangeException for ", STR2 := caseLabel)
		).IsTrue();
	END_IF
END_FOR

accepted := TOF_Core.WideStrings.TryCreateSplitter(
	sourceString := missingSource,
	separator := ",",
	splitter => _Splitter
);
Assert.ThatBool(
	actual := accepted,
	message := "TryCreateSplitter must return FALSE for an unbound source"
).IsFalse();
END_METHOD

(*!
<summary>Verifies that all 80 separator units are used when locating the two fragments.</summary>
<param name="scenario">Factory name included in failure messages.</param>
*)
METHOD PRIVATE assertMaximumSplit
VAR_INPUT
	scenario : WSTRING(80);
END_VAR
VAR
	entry : REFERENCE TO WSTRING;
	advanced : BOOL;
END_VAR
advanced := _Splitter.MoveNext();
entry REF= _Splitter.CurrentEntry;
Assert.ThatBool(
	actual := advanced AND_THEN __ISVALIDREF(entry) AND_THEN entry = "x",
	message := scenario
).IsTrue();

advanced := _Splitter.MoveNext();
entry REF= _Splitter.CurrentEntry;
Assert.ThatBool(
	actual := advanced AND_THEN __ISVALIDREF(entry) AND_THEN entry = "y",
	message := scenario
).IsTrue();

advanced := _Splitter.MoveNext();
Assert.ThatBool(actual := advanced, message := scenario).IsFalse();
END_METHOD

(*!
<summary>Resets the splitter and releases any active fragment before reporting.</summary>
<description>
Safe after partial initialization and after explicit cleanup in the scenario.
</description>
*)
METHOD PROTECTED AfterTest
_Splitter.Reset();
END_METHOD

//! <summary>Borrows the concrete class name. Callers must not modify it.</summary>
{attribute 'monitoring' := 'call'}
PROPERTY ClassName : REFERENCE TO STRING
GET
ClassName REF= _ClassName;
END_GET
END_PROPERTY

//! <summary>Borrows the compiler-initialized namespace name. Callers must not modify it.</summary>
{attribute 'monitoring' := 'call'}
PROPERTY NamespaceName : REFERENCE TO STRING
GET
NamespaceName REF= CurrentNamespace.Name;
END_GET
END_PROPERTY

//! <summary>Reports the concrete instance size in bytes.</summary>
{attribute 'monitoring' := 'call'}
PROPERTY SelfSize : ULINT
GET
SelfSize := XSIZEOF(THIS^);
END_GET
END_PROPERTY

END_FUNCTION_BLOCK

// ---- Tests/Strings/WideString/WideStringLongFitFormattingTest.TcPOU
(*
SPDX-FileCopyrightText: c 2026 Oleksandr Tiutyk <trofimich@gmail.com>
SPDX-License-Identifier: MIT
License: https://opensource.org/license/mit
*)

(*!
<summary>Checks exact 255-unit and truncated 256-unit ANY text formatting.</summary>
<description>
Uses one task and stays at a stable address while assertions are bound to this instance.
</description>
*)

{attribute 'no_assign'}
{attribute 'no_explicit_call' := 'do not call this function block directly'}
FUNCTION_BLOCK WideStringLongFitFormattingTest EXTENDS TOF_Testing.SingleCycleTest
VAR_STAT
	{attribute 'hide'}
	_ClassName : STRING := __POUNAME();
END_VAR

(*!
<summary>Checks exact 255-unit and truncated 256-unit ANY text formatting.</summary>
<description>
Checks the retained code units, the U+2026 marker and the terminator directly in the returned buffer.
</description>
*)
METHOD PROTECTED ExecuteTest
VAR
	narrow : STRING(256);
	wide : WSTRING(256);
	wideData : POINTER TO WORD;
	result : WSTRING(255);
	resultData : POINTER TO WORD;
	i : INT;
END_VAR
wideData := ADR(wide);
resultData := ADR(result);

// SA0175: Fill STRING(256) with 256 ASCII bytes and terminate explicitly.
{analysis -175}
FOR i := 0 TO 255 DO
	narrow[i] := BYTE#16#61;
	wideData[i] := WORD#16#61;
END_FOR

narrow[256] := TO_BYTE(TOF_Core.UnsignedInt8.MIN_VALUE);
{analysis +175}
wideData[256] := TO_WORD(TOF_Core.UnsignedInt16.MIN_VALUE);

result := TOF_Core.WideStrings.AnyToStringFit255(value := narrow);
Assert.ThatBool(
	actual := TOF_Core.WideStrings.GetLength(value := result) = 255
		AND_THEN resultData[253] = WORD#16#61
		AND_THEN resultData[254] = WORD#16#2026
		AND_THEN resultData[255] = TO_WORD(TOF_Core.UnsignedInt16.MIN_VALUE),
	message := "A long STRING must retain 254 characters and append exactly U+2026"
).IsTrue();

result := TOF_Core.WideStrings.AnyToStringFit255(value := wide);
Assert.ThatBool(
	actual := TOF_Core.WideStrings.GetLength(value := result) = 255
		AND_THEN resultData[253] = WORD#16#61
		AND_THEN resultData[254] = WORD#16#2026
		AND_THEN resultData[255] = TO_WORD(TOF_Core.UnsignedInt16.MIN_VALUE),
	message := "A long WSTRING must retain 254 characters and append exactly U+2026"
).IsTrue();

// SA0175: Shorten the ASCII payload to exactly 255 bytes by moving its terminator.
{analysis -175}
narrow[255] := TO_BYTE(TOF_Core.UnsignedInt8.MIN_VALUE);
{analysis +175}
wideData[255] := TO_WORD(TOF_Core.UnsignedInt16.MIN_VALUE);
result := TOF_Core.WideStrings.AnyToStringFit255(value := narrow);
Assert.ThatBool(
	actual := TOF_Core.WideStrings.GetLength(value := result) = 255 AND_THEN resultData[254] = WORD#16#61,
	message := "An exact-fit STRING must keep its final character"
).IsTrue();
result := TOF_Core.WideStrings.AnyToStringFit255(value := wide);
Assert.ThatBool(
	actual := TOF_Core.WideStrings.GetLength(value := result) = 255 AND_THEN resultData[254] = WORD#16#61,
	message := "An exact-fit WSTRING must keep its final character"
).IsTrue();
END_METHOD

//! <summary>Borrows the concrete class name. Callers must not modify it.</summary>
{attribute 'monitoring' := 'call'}
PROPERTY ClassName : REFERENCE TO STRING
GET
ClassName REF= _ClassName;
END_GET
END_PROPERTY

//! <summary>Borrows the compiler-initialized namespace name. Callers must not modify it.</summary>
{attribute 'monitoring' := 'call'}
PROPERTY NamespaceName : REFERENCE TO STRING
GET
NamespaceName REF= CurrentNamespace.Name;
END_GET
END_PROPERTY

//! <summary>Reports the concrete instance size in bytes.</summary>
{attribute 'monitoring' := 'call'}
PROPERTY SelfSize : ULINT
GET
SelfSize := XSIZEOF(THIS^);
END_GET
END_PROPERTY

END_FUNCTION_BLOCK

// ---- Tests/Strings/String/StringBuilderTestGroup.TcPOU
(*
SPDX-FileCopyrightText: c 2026 Oleksandr Tiutyk <trofimich@gmail.com>
SPDX-License-Identifier: MIT
License: https://opensource.org/license/mit
*)

(*!
<summary>Groups byte-string builder assignment, reuse and failure contracts.</summary>
<description>
Owns the independent child instances and their fixed registration array. Use from one PLC task at a stable address.
</description>
*)

{attribute 'no_assign'}
{attribute 'no_explicit_call' := 'do not call this function block directly'}
FUNCTION_BLOCK StringBuilderTestGroup EXTENDS TOF_Testing.TestGroup<3>
VAR_STAT
	{attribute 'hide'}
	_ClassName : STRING := __POUNAME();
END_VAR
VAR
	_BuildEmpty : StringBuilderEmptyTest(name := "BuildEmpty", parent := THIS^);
	_BuildNotEmpty : StringBuilderContentTest(name := "BuildNotEmpty", parent := THIS^);
	_ErrorChecking : StringBuilderAssignmentFailureTest(name := "ErrorChecking", parent := THIS^);

	_Children : ARRAY [0.._ChildCount - 1] OF TOF_Testing.ITestElement :=
	[
		_BuildEmpty,
		_BuildNotEmpty,
		_ErrorChecking
	];
END_VAR

//! <summary>Borrows the fixed child array. Callers must not modify it.</summary>
{attribute 'monitoring' := 'call'}
PROPERTY Children : REFERENCE TO ARRAY [0.._ChildCount - 1] OF TOF_Testing.ITestElement
GET
Children REF= _Children;
END_GET
END_PROPERTY

//! <summary>Borrows the concrete class name. Callers must not modify it.</summary>
{attribute 'monitoring' := 'call'}
PROPERTY ClassName : REFERENCE TO STRING
GET
ClassName REF= _ClassName;
END_GET
END_PROPERTY

//! <summary>Borrows the compiler-initialized namespace name. Callers must not modify it.</summary>
{attribute 'monitoring' := 'call'}
PROPERTY NamespaceName : REFERENCE TO STRING
GET
NamespaceName REF= CurrentNamespace.Name;
END_GET
END_PROPERTY

//! <summary>Reports the concrete instance size in bytes.</summary>
{attribute 'monitoring' := 'call'}
PROPERTY SelfSize : ULINT
GET
SelfSize := XSIZEOF(THIS^);
END_GET
END_PROPERTY

END_FUNCTION_BLOCK

// ---- Tests/Strings/String/StringBuilderEmptyTest.TcPOU
(*
SPDX-FileCopyrightText: c 2026 Oleksandr Tiutyk <trofimich@gmail.com>
SPDX-License-Identifier: MIT
License: https://opensource.org/license/mit
*)

(*!
<summary>Checks assigning an empty builder to a populated target without allocating a builder buffer.</summary>
<description>
Uses one task and stays at a stable address while assertions are bound to this instance.
</description>
*)

{attribute 'no_assign'}
{attribute 'no_explicit_call' := 'do not call this function block directly'}
FUNCTION_BLOCK StringBuilderEmptyTest EXTENDS TOF_Testing.SingleCycleTest
VAR_STAT
	{attribute 'hide'}
	_ClassName : STRING := __POUNAME();
END_VAR
VAR
	_Builder : TOF_Core.StringBuilder;
END_VAR

(*!
<summary>Checks assigning an empty builder to a populated target without allocating a builder buffer.</summary>
<description>
The builder is persistent so teardown can release its buffer after an unexpected hook exception.
</description>
*)
METHOD PROTECTED ExecuteTest
VAR
	target : STRING := 'previous contents';
	copied : BOOL;
END_VAR
copied := _Builder.AssignToString(targetString := target);
Assert.ThatBool(
	actual := copied AND_THEN target = '',
	message := "Assigning an empty builder must clear the target and succeed"
).IsTrue();
Assert.ThatBool(
	actual := _Builder.StringLength = 0 AND_THEN _Builder.Capacity = 0,
	message := "Assigning an empty builder must leave it unallocated"
).IsTrue();
END_METHOD

(*!
<summary>Releases the builder buffer before reporting the case result.</summary>
<description>
Safe after partial initialization and after explicit cleanup in the scenario.
</description>
*)
METHOD PROTECTED AfterTest
_Builder.Clear(releaseMemory := TRUE);
END_METHOD

//! <summary>Borrows the concrete class name. Callers must not modify it.</summary>
{attribute 'monitoring' := 'call'}
PROPERTY ClassName : REFERENCE TO STRING
GET
ClassName REF= _ClassName;
END_GET
END_PROPERTY

//! <summary>Borrows the compiler-initialized namespace name. Callers must not modify it.</summary>
{attribute 'monitoring' := 'call'}
PROPERTY NamespaceName : REFERENCE TO STRING
GET
NamespaceName REF= CurrentNamespace.Name;
END_GET
END_PROPERTY

//! <summary>Reports the concrete instance size in bytes.</summary>
{attribute 'monitoring' := 'call'}
PROPERTY SelfSize : ULINT
GET
SelfSize := XSIZEOF(THIS^);
END_GET
END_PROPERTY

END_FUNCTION_BLOCK

// ---- Tests/Strings/String/StringBuilderContentTest.TcPOU
(*
SPDX-FileCopyrightText: c 2026 Oleksandr Tiutyk <trofimich@gmail.com>
SPDX-License-Identifier: MIT
License: https://opensource.org/license/mit
*)

(*!
<summary>Checks chaining, retained-capacity reuse and a STRING longer than 255 characters.</summary>
<description>
Uses one task and stays at a stable address while assertions are bound to this instance.
</description>
*)

{attribute 'no_assign'}
{attribute 'no_explicit_call' := 'do not call this function block directly'}
FUNCTION_BLOCK StringBuilderContentTest EXTENDS TOF_Testing.SingleCycleTest
VAR_STAT
	{attribute 'hide'}
	_ClassName : STRING := __POUNAME();
END_VAR
VAR
	_Builder : TOF_Core.StringBuilder;
END_VAR

(*!
<summary>Checks chaining, retained-capacity reuse and a STRING longer than 255 characters.</summary>
<description>
The builder is persistent so teardown can release its buffer after an unexpected hook exception.
The 320-byte ASCII fixture and the copied buffer are compared including the terminator.
</description>
*)
METHOD PROTECTED ExecuteTest
VAR
	first : STRING := 'String1';
	second : STRING := 'String2';
	target : STRING(320);
	longText : STRING(320);
	originalBuffer : POINTER TO STRING;
	inputBytes : POINTER TO BYTE;
	outputBytes : POINTER TO BYTE;
	reservedCapacity : UDINT;
	copied : BOOL;
END_VAR
_Builder
	.Append(value := first)
	.AppendIf(value := first, condition := FALSE)
	.AppendString(value := second)
	.AppendStringIf(value := second, condition := FALSE)
	.AppendString255(value := 'String3')
	.AppendString255If(value := 'String3', condition := FALSE);

copied := _Builder.AssignToString(targetString := target);
Assert.ThatBool(
	actual := copied AND_THEN target = 'String1String2String3',
	message := "Chaining must retain all included fragments in order"
).IsTrue();
Assert.ThatUDInt(
	actual := _Builder.StringLength,
	message := "Builder length must exclude the terminator"
).ToBe(expected := UDINT#21);

reservedCapacity := _Builder.Capacity;
originalBuffer := _Builder.StringAddress;
_Builder.Clear(releaseMemory := FALSE);
Assert.ThatBool(
	actual := _Builder.StringLength = 0
		AND_THEN _Builder.Capacity = reservedCapacity
		AND_THEN _Builder.StringAddress = originalBuffer,
	message := "Clear without release must empty the builder while preserving its allocation"
).IsTrue();

copied := _Builder.AssignToString(targetString := target);
Assert.ThatBool(
	actual := copied AND_THEN target = '',
	message := "Clearing the builder must hide the previous text"
).IsTrue();

// SA0175: The 320-byte ASCII fixture needs an exact byte at its last character and a terminator.
{analysis -175}
inputBytes := ADR(longText);
{analysis +175}
Tc2_System.MEMSET(destAddr := inputBytes, fillByte := BYTE#16#61, n := 320);
inputBytes[319] := BYTE#16#7A;
inputBytes[320] := TO_BYTE(TOF_Core.UnsignedInt8.MIN_VALUE);

_Builder.Append(value := longText);
copied := _Builder.AssignToString(targetString := target);

// SA0175: Inspect the bounded byte representation of the ASCII copy, including its terminator.
{analysis -175}
outputBytes := ADR(target);
{analysis +175}
Assert.ThatUDInt(
	actual := _Builder.StringLength,
	message := "Append through ANY must preserve the long STRING length"
).ToBe(expected := UDINT#320);
Assert.ThatBool(
	actual := copied AND_THEN outputBytes[319] = BYTE#16#7A
		AND_THEN outputBytes[320] = TO_BYTE(TOF_Core.UnsignedInt8.MIN_VALUE),
	message := "AssignToString must copy the last byte beyond 255 and its terminator"
).IsTrue();
Assert.ThatBool(
	actual := Tc2_System.MEMCMP(pBuf1 := inputBytes, pBuf2 := outputBytes, n := SIZEOF(target)) = 0,
	message := "The long STRING must round-trip byte for byte"
).IsTrue();

_Builder.Clear(releaseMemory := TRUE);
Assert.ThatBool(
	actual := _Builder.Capacity = 0 AND_THEN _Builder.StringAddress = TOF_Core.Memory.NULL_ADDRESS,
	message := "Clear with release must reset both the capacity and the address"
).IsTrue();
END_METHOD

(*!
<summary>Releases the builder buffer before reporting the case result.</summary>
<description>
Safe after partial initialization and after explicit cleanup in the scenario.
</description>
*)
METHOD PROTECTED AfterTest
_Builder.Clear(releaseMemory := TRUE);
END_METHOD

//! <summary>Borrows the concrete class name. Callers must not modify it.</summary>
{attribute 'monitoring' := 'call'}
PROPERTY ClassName : REFERENCE TO STRING
GET
ClassName REF= _ClassName;
END_GET
END_PROPERTY

//! <summary>Borrows the compiler-initialized namespace name. Callers must not modify it.</summary>
{attribute 'monitoring' := 'call'}
PROPERTY NamespaceName : REFERENCE TO STRING
GET
NamespaceName REF= CurrentNamespace.Name;
END_GET
END_PROPERTY

//! <summary>Reports the concrete instance size in bytes.</summary>
{attribute 'monitoring' := 'call'}
PROPERTY SelfSize : ULINT
GET
SelfSize := XSIZEOF(THIS^);
END_GET
END_PROPERTY

END_FUNCTION_BLOCK

// ---- Tests/Strings/String/StringBuilderAssignmentFailureTest.TcPOU
(*
SPDX-FileCopyrightText: c 2026 Oleksandr Tiutyk <trofimich@gmail.com>
SPDX-License-Identifier: MIT
License: https://opensource.org/license/mit
*)

(*!
<summary>Checks the concrete assignment failures and recovery with a matching buffer.</summary>
<description>
Uses one task and stays at a stable address while assertions are bound to this instance.
</description>
*)

{attribute 'no_assign'}
{attribute 'no_explicit_call' := 'do not call this function block directly'}
FUNCTION_BLOCK StringBuilderAssignmentFailureTest EXTENDS TOF_Testing.SingleCycleTest
VAR_STAT
	{attribute 'hide'}
	_ClassName : STRING := __POUNAME();
END_VAR
VAR
	_Builder : TOF_Core.StringBuilder;
END_VAR

(*!
<summary>Checks the concrete assignment failures and recovery with a matching buffer.</summary>
<description>
The builder is persistent so teardown can release its buffer after an unexpected hook exception.
</description>
*)
METHOD PROTECTED ExecuteTest
VAR
	wideTarget : WSTRING := "wide sentinel";
	shortTarget : STRING(10) := 'keep';
	exactTarget : STRING(16);

	exceptionCode : __SYSTEM.ExceptionCode;
	caught : TOF_Core.IException;
	typeException : TOF_Core.IArgumentTypeClassNotSupportedException;
	capacityException : TOF_Core.ITargetVariableMemoryOverflowException;
	copied : BOOL;
END_VAR
_Builder.AppendString255(value := 'String1234567890');

// Invoke a wrong-width target and check that the argument is rejected before modification.
__TRY
	_Builder.AssignToString(targetString := wideTarget);
__CATCH(exceptionCode)
	caught := TOF_Core.ExceptionManager.GetLastException(
		exceptionCode := exceptionCode,
		catchPointNamespaceName := NamespaceName,
		catchPointPOUName := __POUNAME(),
		catchPointPosition := __POSITION()
	);
__ENDTRY

Assert.ThatBool(
	actual := __QUERYINTERFACE(caught, typeException),
	message := "AssignToString must report an incompatible WSTRING target"
).IsTrue();
Assert.ThatBool(
	actual := wideTarget = "wide sentinel",
	message := "Wrong-width assignment must preserve the target"
).IsTrue();

caught := 0;

// Invoke an undersized STRING target and capture the documented capacity exception.
__TRY
	_Builder.AssignToString(targetString := shortTarget);
__CATCH(exceptionCode)
	caught := TOF_Core.ExceptionManager.GetLastException(
		exceptionCode := exceptionCode,
		catchPointNamespaceName := NamespaceName,
		catchPointPOUName := __POUNAME(),
		catchPointPosition := __POSITION()
	);
__ENDTRY

Assert.ThatBool(
	actual := __QUERYINTERFACE(caught, capacityException),
	message := "AssignToString must report insufficient capacity"
).IsTrue();
Assert.ThatBool(
	actual := shortTarget = 'keep',
	message := "Capacity rejection must preserve the target"
).IsTrue();

copied := _Builder.AssignToString(targetString := exactTarget);
Assert.ThatBool(
	actual := copied AND_THEN exactTarget = 'String1234567890',
	message := "The same builder must still copy successfully into the exact-fit target"
).IsTrue();
END_METHOD

(*!
<summary>Releases the builder buffer before reporting the case result.</summary>
<description>
Safe after partial initialization and after explicit cleanup in the scenario.
</description>
*)
METHOD PROTECTED AfterTest
_Builder.Clear(releaseMemory := TRUE);
END_METHOD

//! <summary>Borrows the concrete class name. Callers must not modify it.</summary>
{attribute 'monitoring' := 'call'}
PROPERTY ClassName : REFERENCE TO STRING
GET
ClassName REF= _ClassName;
END_GET
END_PROPERTY

//! <summary>Borrows the compiler-initialized namespace name. Callers must not modify it.</summary>
{attribute 'monitoring' := 'call'}
PROPERTY NamespaceName : REFERENCE TO STRING
GET
NamespaceName REF= CurrentNamespace.Name;
END_GET
END_PROPERTY

//! <summary>Reports the concrete instance size in bytes.</summary>
{attribute 'monitoring' := 'call'}
PROPERTY SelfSize : ULINT
GET
SelfSize := XSIZEOF(THIS^);
END_GET
END_PROPERTY

END_FUNCTION_BLOCK

// ---- Tests/Strings/WideString/WideStringBuilderTestGroup.TcPOU
(*
SPDX-FileCopyrightText: c 2026 Oleksandr Tiutyk <trofimich@gmail.com>
SPDX-License-Identifier: MIT
License: https://opensource.org/license/mit
*)

(*!
<summary>Groups wide-string builder assignment, reuse and failure cases.</summary>
<description>
Owns the independent child instances and their fixed registration array. Use from one PLC task at a stable address.
</description>
*)

{attribute 'no_assign'}
{attribute 'no_explicit_call' := 'do not call this function block directly'}
FUNCTION_BLOCK WideStringBuilderTestGroup EXTENDS TOF_Testing.TestGroup<3>
VAR_STAT
	{attribute 'hide'}
	_ClassName : STRING := __POUNAME();
END_VAR
VAR
	_BuildEmpty : WideStringBuilderEmptyTest(name := "BuildEmpty", parent := THIS^);
	_BuildNotEmpty : WideStringBuilderContentTest(name := "BuildNotEmpty", parent := THIS^);
	_ErrorChecking : WideStringBuilderAssignmentFailureTest(name := "ErrorChecking", parent := THIS^);

	_Children : ARRAY [0.._ChildCount - 1] OF TOF_Testing.ITestElement :=
	[
		_BuildEmpty,
		_BuildNotEmpty,
		_ErrorChecking
	];
END_VAR

//! <summary>Borrows the fixed child array. Callers must not modify it.</summary>
{attribute 'monitoring' := 'call'}
PROPERTY Children : REFERENCE TO ARRAY [0.._ChildCount - 1] OF TOF_Testing.ITestElement
GET
Children REF= _Children;
END_GET
END_PROPERTY

//! <summary>Borrows the concrete class name. Callers must not modify it.</summary>
{attribute 'monitoring' := 'call'}
PROPERTY ClassName : REFERENCE TO STRING
GET
ClassName REF= _ClassName;
END_GET
END_PROPERTY

//! <summary>Borrows the compiler-initialized namespace name. Callers must not modify it.</summary>
{attribute 'monitoring' := 'call'}
PROPERTY NamespaceName : REFERENCE TO STRING
GET
NamespaceName REF= CurrentNamespace.Name;
END_GET
END_PROPERTY

//! <summary>Reports the concrete instance size in bytes.</summary>
{attribute 'monitoring' := 'call'}
PROPERTY SelfSize : ULINT
GET
SelfSize := XSIZEOF(THIS^);
END_GET
END_PROPERTY

END_FUNCTION_BLOCK

// ---- Tests/Strings/WideString/WideStringBuilderEmptyTest.TcPOU
(*
SPDX-FileCopyrightText: c 2026 Oleksandr Tiutyk <trofimich@gmail.com>
SPDX-License-Identifier: MIT
License: https://opensource.org/license/mit
*)

(*!
<summary>Checks assigning an empty builder to a populated target without allocating a builder buffer.</summary>
<description>
Uses one task and stays at a stable address while assertions are bound to this instance.
</description>
*)

{attribute 'no_assign'}
{attribute 'no_explicit_call' := 'do not call this function block directly'}
FUNCTION_BLOCK WideStringBuilderEmptyTest EXTENDS TOF_Testing.SingleCycleTest
VAR_STAT
	{attribute 'hide'}
	_ClassName : STRING := __POUNAME();
END_VAR
VAR
	_Builder : TOF_Core.WideStringBuilder;
END_VAR

(*!
<summary>Checks assigning an empty builder to a populated target without allocating a builder buffer.</summary>
<description>
The builder is persistent so teardown can release its buffer after an unexpected hook exception.
</description>
*)
METHOD PROTECTED ExecuteTest
VAR
	target : WSTRING := "previous contents";
	copied : BOOL;
END_VAR
copied := _Builder.AssignToString(targetString := target);
Assert.ThatBool(
	actual := copied AND_THEN target = "",
	message := "Assigning an empty builder must clear the target and succeed"
).IsTrue();
Assert.ThatBool(
	actual := _Builder.StringLength = 0 AND_THEN _Builder.Capacity = 0,
	message := "Assigning an empty builder must leave it unallocated"
).IsTrue();
END_METHOD

(*!
<summary>Releases the builder buffer before reporting the case result.</summary>
<description>
Safe after partial initialization and after explicit cleanup in the scenario.
</description>
*)
METHOD PROTECTED AfterTest
_Builder.Clear(releaseMemory := TRUE);
END_METHOD

//! <summary>Borrows the concrete class name. Callers must not modify it.</summary>
{attribute 'monitoring' := 'call'}
PROPERTY ClassName : REFERENCE TO STRING
GET
ClassName REF= _ClassName;
END_GET
END_PROPERTY

//! <summary>Borrows the compiler-initialized namespace name. Callers must not modify it.</summary>
{attribute 'monitoring' := 'call'}
PROPERTY NamespaceName : REFERENCE TO STRING
GET
NamespaceName REF= CurrentNamespace.Name;
END_GET
END_PROPERTY

//! <summary>Reports the concrete instance size in bytes.</summary>
{attribute 'monitoring' := 'call'}
PROPERTY SelfSize : ULINT
GET
SelfSize := XSIZEOF(THIS^);
END_GET
END_PROPERTY

END_FUNCTION_BLOCK

// ---- Tests/Strings/WideString/WideStringBuilderContentTest.TcPOU
(*
SPDX-FileCopyrightText: c 2026 Oleksandr Tiutyk <trofimich@gmail.com>
SPDX-License-Identifier: MIT
License: https://opensource.org/license/mit
*)

(*!
<summary>Checks chaining, retained-capacity reuse and a WSTRING longer than 255 characters.</summary>
<description>
Uses one task and stays at a stable address while assertions are bound to this instance.
</description>
*)

{attribute 'no_assign'}
{attribute 'no_explicit_call' := 'do not call this function block directly'}
FUNCTION_BLOCK WideStringBuilderContentTest EXTENDS TOF_Testing.SingleCycleTest
VAR_STAT
	{attribute 'hide'}
	_ClassName : STRING := __POUNAME();
END_VAR
VAR
	_Builder : TOF_Core.WideStringBuilder;
END_VAR

(*!
<summary>Checks chaining, retained-capacity reuse and a WSTRING longer than 255 characters.</summary>
<description>
The builder is persistent so teardown can release its buffer after an unexpected hook exception.
The 320-unit wide fixture and the copied buffer are compared including the terminator.
</description>
*)
METHOD PROTECTED ExecuteTest
VAR
	first : WSTRING := "String1";
	second : WSTRING := "String2";
	target : WSTRING(320);
	longText : WSTRING(320);
	originalBuffer : POINTER TO WSTRING;
	inputUnits : POINTER TO WORD;
	outputUnits : POINTER TO WORD;
	reservedCapacity : UDINT;
	i : DINT;
	copied : BOOL;
END_VAR
_Builder
	.Append(value := first)
	.AppendIf(value := first, condition := FALSE)
	.AppendString(value := second)
	.AppendStringIf(value := second, condition := FALSE)
	.AppendString255(value := "String3")
	.AppendString255If(value := "String3", condition := FALSE);

copied := _Builder.AssignToString(targetString := target);
Assert.ThatBool(
	actual := copied AND_THEN target = "String1String2String3",
	message := "Chaining must retain all included fragments in order"
).IsTrue();
Assert.ThatUDInt(
	actual := _Builder.StringLength,
	message := "Builder length must exclude the terminator"
).ToBe(expected := UDINT#21);

reservedCapacity := _Builder.Capacity;
originalBuffer := _Builder.StringAddress;
_Builder.Clear(releaseMemory := FALSE);
Assert.ThatBool(
	actual := _Builder.StringLength = 0
		AND_THEN _Builder.Capacity = reservedCapacity
		AND_THEN _Builder.StringAddress = originalBuffer,
	message := "Clear without release must empty the builder while preserving its allocation"
).IsTrue();

copied := _Builder.AssignToString(targetString := target);
Assert.ThatBool(
	actual := copied AND_THEN target = "",
	message := "Clearing the builder must hide the previous text"
).IsTrue();

// SA0175: The 320-unit wide fixture needs an exact final code unit and a terminator.
{analysis -175}
inputUnits := ADR(longText);
{analysis +175}

FOR i := 0 TO 318 DO
	inputUnits[i] := WORD#16#0410;
END_FOR

inputUnits[319] := WORD#16#2026;
inputUnits[320] := WORD#0;

// SA0175: Seed the last destination code unit to verify that the copy writes the terminator.
{analysis -175}
outputUnits := ADR(target);
outputUnits[320] := WORD#16#0058;
{analysis +175}

_Builder.Append(value := longText);
copied := _Builder.AssignToString(targetString := target);

Assert.ThatUDInt(
	actual := _Builder.StringLength,
	message := "Append through ANY must preserve the long WSTRING length"
).ToBe(expected := UDINT#320);
Assert.ThatBool(
	actual := copied AND_THEN outputUnits[319] = WORD#16#2026
		AND_THEN outputUnits[320] = WORD#0,
	message := "AssignToString must copy the last code unit beyond 255 and its terminator"
).IsTrue();
Assert.ThatBool(
	actual := Tc2_System.MEMCMP(pBuf1 := inputUnits, pBuf2 := outputUnits, n := SIZEOF(target)) = 0,
	message := "The long WSTRING must round-trip byte for byte"
).IsTrue();

_Builder.Clear(releaseMemory := TRUE);
Assert.ThatBool(
	actual := _Builder.Capacity = 0 AND_THEN _Builder.StringAddress = TOF_Core.Memory.NULL_ADDRESS,
	message := "Clear with release must reset both the capacity and the address"
).IsTrue();
END_METHOD

(*!
<summary>Releases the builder buffer before reporting the case result.</summary>
<description>
Safe after partial initialization and after explicit cleanup in the scenario.
</description>
*)
METHOD PROTECTED AfterTest
_Builder.Clear(releaseMemory := TRUE);
END_METHOD

//! <summary>Borrows the concrete class name. Callers must not modify it.</summary>
{attribute 'monitoring' := 'call'}
PROPERTY ClassName : REFERENCE TO STRING
GET
ClassName REF= _ClassName;
END_GET
END_PROPERTY

//! <summary>Borrows the compiler-initialized namespace name. Callers must not modify it.</summary>
{attribute 'monitoring' := 'call'}
PROPERTY NamespaceName : REFERENCE TO STRING
GET
NamespaceName REF= CurrentNamespace.Name;
END_GET
END_PROPERTY

//! <summary>Reports the concrete instance size in bytes.</summary>
{attribute 'monitoring' := 'call'}
PROPERTY SelfSize : ULINT
GET
SelfSize := XSIZEOF(THIS^);
END_GET
END_PROPERTY

END_FUNCTION_BLOCK

// ---- Tests/Strings/WideString/WideStringBuilderAssignmentFailureTest.TcPOU
(*
SPDX-FileCopyrightText: c 2026 Oleksandr Tiutyk <trofimich@gmail.com>
SPDX-License-Identifier: MIT
License: https://opensource.org/license/mit
*)

(*!
<summary>Checks the concrete assignment failures and recovery with a matching buffer.</summary>
<description>
Uses one task and stays at a stable address while assertions are bound to this instance.
</description>
*)

{attribute 'no_assign'}
{attribute 'no_explicit_call' := 'do not call this function block directly'}
FUNCTION_BLOCK WideStringBuilderAssignmentFailureTest EXTENDS TOF_Testing.SingleCycleTest
VAR_STAT
	{attribute 'hide'}
	_ClassName : STRING := __POUNAME();
END_VAR
VAR
	_Builder : TOF_Core.WideStringBuilder;
END_VAR

(*!
<summary>Checks the concrete assignment failures and recovery with a matching buffer.</summary>
<description>
The builder is persistent so teardown can release its buffer after an unexpected hook exception.
</description>
*)
METHOD PROTECTED ExecuteTest
VAR
	byteTarget : STRING := 'byte sentinel';
	shortTarget : WSTRING(10) := "keep";
	exactTarget : WSTRING(16);

	exceptionCode : __SYSTEM.ExceptionCode;
	caught : TOF_Core.IException;
	typeException : TOF_Core.IArgumentTypeClassNotSupportedException;
	capacityException : TOF_Core.ITargetVariableMemoryOverflowException;
	copied : BOOL;
END_VAR
_Builder.AppendString255(value := "String1234567890");

// Invoke a wrong-width target and check that the argument is rejected before modification.
__TRY
	_Builder.AssignToString(targetString := byteTarget);
__CATCH(exceptionCode)
	caught := TOF_Core.ExceptionManager.GetLastException(
		exceptionCode := exceptionCode,
		catchPointNamespaceName := NamespaceName,
		catchPointPOUName := __POUNAME(),
		catchPointPosition := __POSITION()
	);
__ENDTRY

Assert.ThatBool(
	actual := __QUERYINTERFACE(caught, typeException),
	message := "AssignToString must report an incompatible STRING target"
).IsTrue();
Assert.ThatBool(
	actual := byteTarget = 'byte sentinel',
	message := "Wrong-width assignment must preserve the target"
).IsTrue();

caught := 0;

// Invoke an undersized WSTRING target and capture the documented capacity exception.
__TRY
	_Builder.AssignToString(targetString := shortTarget);
__CATCH(exceptionCode)
	caught := TOF_Core.ExceptionManager.GetLastException(
		exceptionCode := exceptionCode,
		catchPointNamespaceName := NamespaceName,
		catchPointPOUName := __POUNAME(),
		catchPointPosition := __POSITION()
	);
__ENDTRY

Assert.ThatBool(
	actual := __QUERYINTERFACE(caught, capacityException),
	message := "AssignToString must report insufficient capacity"
).IsTrue();
Assert.ThatBool(
	actual := shortTarget = "keep",
	message := "Capacity rejection must preserve the target"
).IsTrue();

copied := _Builder.AssignToString(targetString := exactTarget);
Assert.ThatBool(
	actual := copied AND_THEN exactTarget = "String1234567890",
	message := "The same builder must still copy successfully into the exact-fit target"
).IsTrue();
END_METHOD

(*!
<summary>Releases the builder buffer before reporting the case result.</summary>
<description>
Safe after partial initialization and after explicit cleanup in the scenario.
</description>
*)
METHOD PROTECTED AfterTest
_Builder.Clear(releaseMemory := TRUE);
END_METHOD

//! <summary>Borrows the concrete class name. Callers must not modify it.</summary>
{attribute 'monitoring' := 'call'}
PROPERTY ClassName : REFERENCE TO STRING
GET
ClassName REF= _ClassName;
END_GET
END_PROPERTY

//! <summary>Borrows the compiler-initialized namespace name. Callers must not modify it.</summary>
{attribute 'monitoring' := 'call'}
PROPERTY NamespaceName : REFERENCE TO STRING
GET
NamespaceName REF= CurrentNamespace.Name;
END_GET
END_PROPERTY

//! <summary>Reports the concrete instance size in bytes.</summary>
{attribute 'monitoring' := 'call'}
PROPERTY SelfSize : ULINT
GET
SelfSize := XSIZEOF(THIS^);
END_GET
END_PROPERTY

END_FUNCTION_BLOCK

// ---- Tests/Collections/Dynamic/DynamicByteListTestGroup.TcPOU
(*
SPDX-FileCopyrightText: c 2026 Oleksandr Tiutyk <trofimich@gmail.com>
SPDX-License-Identifier: MIT
License: https://opensource.org/license/mit
*)

(*!
<summary>Groups byte-list operations with dynamically allocated storage.</summary>
<description>
Owns the independent child instances and their fixed registration array. Use from one PLC task at a stable address.
</description>
*)

{attribute 'no_assign'}
{attribute 'no_explicit_call' := 'do not call this function block directly'}
FUNCTION_BLOCK DynamicByteListTestGroup EXTENDS TOF_Testing.TestGroup<6>
VAR_STAT
	{attribute 'hide'}
	_ClassName : STRING := __POUNAME();
END_VAR
VAR
	_LoadFromAny : ByteListLoadFromAnyTest(name := "LoadFromAny", parent := THIS^, useDynamicStorage := TRUE);
	_GetAndSet : ByteListIndexedAccessTest(name := "GetAndSet", parent := THIS^, useDynamicStorage := TRUE);
	_Find : ByteListFindTest(name := "Find", parent := THIS^, useDynamicStorage := TRUE);
	_Remove : ByteListRemoveValueTest(name := "Remove", parent := THIS^, useDynamicStorage := TRUE);
	_RemoveAt : ByteListRemoveRangeTest(name := "RemoveAt", parent := THIS^, useDynamicStorage := TRUE);
	_Clear : ByteListClearTest(name := "Clear", parent := THIS^, useDynamicStorage := TRUE);

	_Children : ARRAY [0.._ChildCount - 1] OF TOF_Testing.ITestElement :=
	[
		_LoadFromAny,
		_GetAndSet,
		_Find,
		_Remove,
		_RemoveAt,
		_Clear
	];
END_VAR

//! <summary>Borrows the fixed child array. Callers must not modify it.</summary>
{attribute 'monitoring' := 'call'}
PROPERTY Children : REFERENCE TO ARRAY [0.._ChildCount - 1] OF TOF_Testing.ITestElement
GET
Children REF= _Children;
END_GET
END_PROPERTY

//! <summary>Borrows the concrete class name. Callers must not modify it.</summary>
{attribute 'monitoring' := 'call'}
PROPERTY ClassName : REFERENCE TO STRING
GET
ClassName REF= _ClassName;
END_GET
END_PROPERTY

//! <summary>Borrows the compiler-initialized namespace name. Callers must not modify it.</summary>
{attribute 'monitoring' := 'call'}
PROPERTY NamespaceName : REFERENCE TO STRING
GET
NamespaceName REF= CurrentNamespace.Name;
END_GET
END_PROPERTY

//! <summary>Reports the concrete instance size in bytes.</summary>
{attribute 'monitoring' := 'call'}
PROPERTY SelfSize : ULINT
GET
SelfSize := XSIZEOF(THIS^);
END_GET
END_PROPERTY

END_FUNCTION_BLOCK

// ---- Tests/Collections/ByteListLoadFromAnyTest.TcPOU
(*
SPDX-FileCopyrightText: c 2026 Oleksandr Tiutyk <trofimich@gmail.com>
SPDX-License-Identifier: MIT
License: https://opensource.org/license/mit
*)

(*!
<summary>Checks byte ordering and end-position loading through ANY.</summary>
<description>
Runs against the selected fixture. The base case clears it before publishing the result.
</description>
*)

{attribute 'no_assign'}
{attribute 'no_explicit_call' := 'do not call this function block directly'}
FUNCTION_BLOCK ByteListLoadFromAnyTest EXTENDS ByteListTestCase
VAR_STAT
	{attribute 'hide'}
	_ClassName : STRING := __POUNAME();
END_VAR

(*!
<summary>Checks byte ordering and end-position loading through ANY.</summary>
*)
METHOD PROTECTED ExecuteTest
VAR
	values : ARRAY [0..5] OF BYTE := [0, 1, 2, 3, 4, 5];
	i : DINT;
END_VAR
_List.LoadFromAny(data := values, startIndex := 0);

Assert.ThatDInt(
	actual := _List.Length,
	message := "Initial load must copy six bytes"
).ToBe(expected := DINT#6);

_List.LoadFromAny(data := values, startIndex := _List.Length);

Assert.ThatDInt(
	actual := _List.Length,
	message := "Loading at the end must extend the list"
).ToBe(expected := DINT#12);

FOR i := 0 TO 11 DO
	Assert.ThatBool(
		actual := _List.Get(index := i) = values[i MOD 6],
		message := "The concatenated buffers must preserve byte order"
	).IsTrue();
END_FOR

_List.LoadFromAny(data := values, startIndex := 2);

Assert.ThatDInt(
	actual := _List.Length,
	message := "A load inside the list must truncate bytes beyond its new end"
).ToBe(expected := DINT#8);

Assert.ThatBool(
	actual := _List.Get(index := 1) = BYTE#1
		AND_THEN _List.Get(index := 2) = BYTE#0
		AND_THEN _List.Get(index := 7) = BYTE#5,
	message := "The partial load must preserve the prefix and write through its final byte"
).IsTrue();
END_METHOD

//! <summary>Borrows the concrete class name. Callers must not modify it.</summary>
{attribute 'monitoring' := 'call'}
PROPERTY ClassName : REFERENCE TO STRING
GET
ClassName REF= _ClassName;
END_GET
END_PROPERTY

//! <summary>Borrows the compiler-initialized namespace name. Callers must not modify it.</summary>
{attribute 'monitoring' := 'call'}
PROPERTY NamespaceName : REFERENCE TO STRING
GET
NamespaceName REF= CurrentNamespace.Name;
END_GET
END_PROPERTY

//! <summary>Reports the concrete instance size in bytes.</summary>
{attribute 'monitoring' := 'call'}
PROPERTY SelfSize : ULINT
GET
SelfSize := XSIZEOF(THIS^);
END_GET
END_PROPERTY

END_FUNCTION_BLOCK

// ---- Tests/Collections/ByteListTestCase.TcPOU
(*
SPDX-FileCopyrightText: c 2026 Oleksandr Tiutyk <trofimich@gmail.com>
SPDX-License-Identifier: MIT
License: https://opensource.org/license/mit
*)

(*!
<summary>Supplies independent byte-list storage and teardown for a single-cycle test.</summary>
<description>
Each case owns concrete dynamic and inline fixtures at a stable address. The constructor selects one fixture.
BeforeTest binds that fixture and AfterTest clears it before the result is published. Descendants supply
ExecuteTest and use the selected list only during that hook. Run each instance from one task.
</description>
*)

{attribute 'no_assign'}
{attribute 'no_explicit_call' := 'do not call this function block directly'}
FUNCTION_BLOCK ABSTRACT ByteListTestCase EXTENDS TOF_Testing.SingleCycleTest
VAR
	//! <summary>Selected storage mode established by FB_init.</summary>
	_UseDynamicStorage : BOOL;
	//! <summary>Borrowed interface to the selected fixture during case execution.</summary>
	_List : TOF_Collections.IByteList;

	_DynamicList : TOF_Collections.ByteList<0>;
	_InlineList : TOF_Collections.ByteList<12>;
END_VAR

(*!
<summary>Selects the storage fixture for the lifetime of the test case.</summary>
<description>Stores only the mode. TestElement initializes the name and parent.</description>
<param name="name">Display name of this case.</param>
<param name="parent">Group that owns this case.</param>
<param name="useDynamicStorage">TRUE selects dynamic storage. FALSE selects the 12-byte inline fixture.</param>
*)
METHOD FB_init : BOOL
VAR_INPUT
	bInitRetains: BOOL; // TRUE: the retain variables are initialized (reset warm / reset cold)
	bInCopyCode: BOOL; // TRUE: the instance will be copied to the copy code afterward (online change)
	name : WSTRING;
	parent : TOF_Testing.ITestElement;
	useDynamicStorage : BOOL;
END_VAR
_UseDynamicStorage := useDynamicStorage;
FB_init := TRUE;
END_METHOD

(*!
<summary>Binds the case to its selected byte-list fixture for the run.</summary>
*)
METHOD PROTECTED FINAL BeforeTest
IF _UseDynamicStorage THEN
	_List := _DynamicList;
ELSE
	_List := _InlineList;
END_IF
END_METHOD

(*!
<summary>Clears the bound fixture and releases dynamic capacity before result publication.</summary>
<description>Accepts a missing binding after interrupted preparation and clears the borrowed interface after use.</description>
*)
METHOD PROTECTED FINAL AfterTest
IF _List <> 0 THEN
	_List.Clear(releaseDynamicMemory := TRUE);
	_List := 0;
END_IF
END_METHOD

(*!
<summary>Borrows the data address of the selected fixture.</summary>
<description>Read again after growth or release. The returned pointer may have become invalid.</description>
*)
METHOD PROTECTED FINAL GetBufferAddress : POINTER TO BYTE
IF _UseDynamicStorage THEN
	GetBufferAddress := _DynamicList.DataAddress;
ELSE
	GetBufferAddress := _InlineList.DataAddress;
END_IF
END_METHOD

END_FUNCTION_BLOCK

// ---- Tests/Collections/ByteListIndexedAccessTest.TcPOU
(*
SPDX-FileCopyrightText: c 2026 Oleksandr Tiutyk <trofimich@gmail.com>
SPDX-License-Identifier: MIT
License: https://opensource.org/license/mit
*)

(*!
<summary>Checks appended bytes, replacement and rejected Set indices.</summary>
<description>
Runs against the selected fixture. The base case clears it before publishing the result.
</description>
*)

{attribute 'no_assign'}
{attribute 'no_explicit_call' := 'do not call this function block directly'}
FUNCTION_BLOCK ByteListIndexedAccessTest EXTENDS ByteListTestCase
VAR_STAT
	{attribute 'hide'}
	_ClassName : STRING := __POUNAME();
END_VAR

(*!
<summary>Checks appended bytes, replacement and rejected Set indices.</summary>
*)
METHOD PROTECTED ExecuteTest
VAR
	values : ARRAY [0..5] OF BYTE := [0, 1, 2, 3, 4, 5];
	i : DINT;
	invalidIndex : DINT;

	exceptionCode : __SYSTEM.ExceptionCode;
	caught : TOF_Core.IException;
	standardException : TOF_Core.IStandardException;
	message : TOF_Core.ERROR_MESSAGE;
END_VAR
FOR i := 0 TO 5 DO
	_List.AppendByte(value := values[i]);
END_FOR

_List.AppendAny(data := values);

FOR i := 0 TO 11 DO
	Assert.ThatBool(
		actual := _List.Get(index := i) = values[i MOD 6],
		message := "AppendByte and AppendAny must preserve the input bytes"
	).IsTrue();
END_FOR

_List.Set(index := 5, value := BYTE#50);

Assert.ThatBool(
	actual := _List.Get(index := 5) = BYTE#50,
	message := "Set must replace the requested byte"
).IsTrue();

// Pass the invalid value at runtime so Set can exercise its negative-index guard.
invalidIndex := -1;

__TRY
	_List.Set(index := invalidIndex, value := BYTE#10);
__CATCH(exceptionCode)
	caught := TOF_Core.ExceptionManager.GetLastException(
		exceptionCode := exceptionCode,
		catchPointNamespaceName := NamespaceName,
		catchPointPOUName := __POUNAME(),
		catchPointPosition := __POSITION()
	);
__ENDTRY

Assert.ThatBool(
	actual := __QUERYINTERFACE(caught, standardException),
	message := "Set at index -1 must raise StandardException"
).IsTrue();

IF caught <> 0 THEN
	message := caught.GetMessage();
	Assert.ThatBool(
		actual := message = "Index is less then zero",
		message := "Set at index -1 must identify the violated bound"
	).IsTrue();
END_IF

Assert.ThatDInt(
	actual := _List.Length,
	message := "Set at index -1 must preserve length"
).ToBe(expected := DINT#12);

Assert.ThatBool(
	actual := _List.Get(index := 5) = BYTE#50,
	message := "Set at index -1 must preserve the replaced byte"
).IsTrue();

caught := 0;

__TRY
	_List.Set(index := 12, value := BYTE#10);
__CATCH(exceptionCode)
	caught := TOF_Core.ExceptionManager.GetLastException(
		exceptionCode := exceptionCode,
		catchPointNamespaceName := NamespaceName,
		catchPointPOUName := __POUNAME(),
		catchPointPosition := __POSITION()
	);
__ENDTRY

Assert.ThatBool(
	actual := __QUERYINTERFACE(caught, standardException),
	message := "Set at index 12 must raise StandardException"
).IsTrue();

IF caught <> 0 THEN
	message := caught.GetMessage();
	Assert.ThatBool(
		actual := message = "Index is too large",
		message := "Set at index 12 must identify the violated bound"
	).IsTrue();
END_IF

Assert.ThatDInt(
	actual := _List.Length,
	message := "Set at index 12 must preserve length"
).ToBe(expected := DINT#12);

Assert.ThatBool(
	actual := _List.Get(index := 5) = BYTE#50,
	message := "Set at index 12 must preserve the replaced byte"
).IsTrue();
END_METHOD

//! <summary>Borrows the concrete class name. Callers must not modify it.</summary>
{attribute 'monitoring' := 'call'}
PROPERTY ClassName : REFERENCE TO STRING
GET
ClassName REF= _ClassName;
END_GET
END_PROPERTY

//! <summary>Borrows the compiler-initialized namespace name. Callers must not modify it.</summary>
{attribute 'monitoring' := 'call'}
PROPERTY NamespaceName : REFERENCE TO STRING
GET
NamespaceName REF= CurrentNamespace.Name;
END_GET
END_PROPERTY

//! <summary>Reports the concrete instance size in bytes.</summary>
{attribute 'monitoring' := 'call'}
PROPERTY SelfSize : ULINT
GET
SelfSize := XSIZEOF(THIS^);
END_GET
END_PROPERTY

END_FUNCTION_BLOCK

// ---- Tests/Collections/ByteListFindTest.TcPOU
(*
SPDX-FileCopyrightText: c 2026 Oleksandr Tiutyk <trofimich@gmail.com>
SPDX-License-Identifier: MIT
License: https://opensource.org/license/mit
*)

(*!
<summary>Checks the first match and absence without changing the byte list.</summary>
<description>
Runs against the selected fixture. The base case clears it before publishing the result.
</description>
*)

{attribute 'no_assign'}
{attribute 'no_explicit_call' := 'do not call this function block directly'}
FUNCTION_BLOCK ByteListFindTest EXTENDS ByteListTestCase
VAR_STAT
	{attribute 'hide'}
	_ClassName : STRING := __POUNAME();
END_VAR

(*!
<summary>Checks the first match and absence without changing the byte list.</summary>
*)
METHOD PROTECTED ExecuteTest
VAR
	values : ARRAY [0..5] OF BYTE := [0, 1, 2, 3, 4, 5];
	found : BOOL;
	index : DINT;
END_VAR
_List.AppendAny(data := values);
_List.Set(index := 5, value := BYTE#50);

found := _List.Find(value := BYTE#50, index => index);

Assert.ThatBool(
	actual := found AND_THEN index = 5,
	message := "Find must return the replaced byte at index 5"
).IsTrue();

_List.AppendByte(value := BYTE#50);

found := _List.Find(value := BYTE#50, index => index);

Assert.ThatBool(
	actual := found AND_THEN index = 5,
	message := "Find must select the first duplicate"
).IsTrue();

found := _List.Find(value := BYTE#255, index => index);

Assert.ThatBool(
	actual := NOT found,
	message := "Find must report absence for an unmatched byte"
).IsTrue();
END_METHOD

//! <summary>Borrows the concrete class name. Callers must not modify it.</summary>
{attribute 'monitoring' := 'call'}
PROPERTY ClassName : REFERENCE TO STRING
GET
ClassName REF= _ClassName;
END_GET
END_PROPERTY

//! <summary>Borrows the compiler-initialized namespace name. Callers must not modify it.</summary>
{attribute 'monitoring' := 'call'}
PROPERTY NamespaceName : REFERENCE TO STRING
GET
NamespaceName REF= CurrentNamespace.Name;
END_GET
END_PROPERTY

//! <summary>Reports the concrete instance size in bytes.</summary>
{attribute 'monitoring' := 'call'}
PROPERTY SelfSize : ULINT
GET
SelfSize := XSIZEOF(THIS^);
END_GET
END_PROPERTY

END_FUNCTION_BLOCK

// ---- Tests/Collections/ByteListRemoveValueTest.TcPOU
(*
SPDX-FileCopyrightText: c 2026 Oleksandr Tiutyk <trofimich@gmail.com>
SPDX-License-Identifier: MIT
License: https://opensource.org/license/mit
*)

(*!
<summary>Checks first-match removal and preservation on a missing value.</summary>
<description>
Runs against the selected fixture. The base case clears it before publishing the result.
</description>
*)

{attribute 'no_assign'}
{attribute 'no_explicit_call' := 'do not call this function block directly'}
FUNCTION_BLOCK ByteListRemoveValueTest EXTENDS ByteListTestCase
VAR_STAT
	{attribute 'hide'}
	_ClassName : STRING := __POUNAME();
END_VAR

(*!
<summary>Checks first-match removal and preservation on a missing value.</summary>
*)
METHOD PROTECTED ExecuteTest
VAR
	expected : ARRAY [0..4] OF BYTE := [1, 3, 2, 4, 5];
	values : ARRAY [0..5] OF BYTE := [1, 2, 3, 2, 4, 5];
	i : DINT;
END_VAR
_List.AppendAny(data := values);
_List.Remove(value := BYTE#2);

Assert.ThatDInt(
	actual := _List.Length,
	message := "Remove must remove one matching byte"
).ToBe(expected := DINT#5);

_List.Remove(value := BYTE#255);

Assert.ThatDInt(
	actual := _List.Length,
	message := "Removing a missing byte must preserve length"
).ToBe(expected := DINT#5);

FOR i := 0 TO 4 DO
	Assert.ThatBool(
		actual := _List.Get(index := i) = expected[i],
		message := "Removal must preserve survivors in order"
	).IsTrue();
END_FOR
END_METHOD

//! <summary>Borrows the concrete class name. Callers must not modify it.</summary>
{attribute 'monitoring' := 'call'}
PROPERTY ClassName : REFERENCE TO STRING
GET
ClassName REF= _ClassName;
END_GET
END_PROPERTY

//! <summary>Borrows the compiler-initialized namespace name. Callers must not modify it.</summary>
{attribute 'monitoring' := 'call'}
PROPERTY NamespaceName : REFERENCE TO STRING
GET
NamespaceName REF= CurrentNamespace.Name;
END_GET
END_PROPERTY

//! <summary>Reports the concrete instance size in bytes.</summary>
{attribute 'monitoring' := 'call'}
PROPERTY SelfSize : ULINT
GET
SelfSize := XSIZEOF(THIS^);
END_GET
END_PROPERTY

END_FUNCTION_BLOCK

// ---- Tests/Collections/ByteListRemoveRangeTest.TcPOU
(*
SPDX-FileCopyrightText: c 2026 Oleksandr Tiutyk <trofimich@gmail.com>
SPDX-License-Identifier: MIT
License: https://opensource.org/license/mit
*)

(*!
<summary>Checks middle-range compaction and exact suffix deletion.</summary>
<description>
Runs against the selected fixture. The base case clears it before publishing the result.
</description>
*)

{attribute 'no_assign'}
{attribute 'no_explicit_call' := 'do not call this function block directly'}
FUNCTION_BLOCK ByteListRemoveRangeTest EXTENDS ByteListTestCase
VAR_STAT
	{attribute 'hide'}
	_ClassName : STRING := __POUNAME();
END_VAR

(*!
<summary>Checks middle-range compaction and exact suffix deletion.</summary>
*)
METHOD PROTECTED ExecuteTest
VAR
	values : ARRAY [0..5] OF BYTE := [0, 1, 2, 3, 4, 5];
	expected : ARRAY [0..3] OF BYTE := [0, 1, 4, 5];
	i : DINT;
END_VAR
_List.AppendAny(data := values);
_List.RemoveAt(index := 2, count := 2);

Assert.ThatDInt(
	actual := _List.Length,
	message := "Removing two middle bytes must leave four bytes"
).ToBe(expected := DINT#4);

FOR i := 0 TO 3 DO
	Assert.ThatBool(
		actual := _List.Get(index := i) = expected[i],
		message := "The remaining bytes must stay in order"
	).IsTrue();
END_FOR

_List.RemoveAt(index := 2, count := 2);

Assert.ThatDInt(
	actual := _List.Length,
	message := "Removing through the end must preserve the prefix length"
).ToBe(expected := DINT#2);

Assert.ThatBool(
	actual := _List.Get(index := 0) = BYTE#0 AND_THEN _List.Get(index := 1) = BYTE#1,
	message := "Removing the suffix must preserve the prefix bytes"
).IsTrue();
END_METHOD

//! <summary>Borrows the concrete class name. Callers must not modify it.</summary>
{attribute 'monitoring' := 'call'}
PROPERTY ClassName : REFERENCE TO STRING
GET
ClassName REF= _ClassName;
END_GET
END_PROPERTY

//! <summary>Borrows the compiler-initialized namespace name. Callers must not modify it.</summary>
{attribute 'monitoring' := 'call'}
PROPERTY NamespaceName : REFERENCE TO STRING
GET
NamespaceName REF= CurrentNamespace.Name;
END_GET
END_PROPERTY

//! <summary>Reports the concrete instance size in bytes.</summary>
{attribute 'monitoring' := 'call'}
PROPERTY SelfSize : ULINT
GET
SelfSize := XSIZEOF(THIS^);
END_GET
END_PROPERTY

END_FUNCTION_BLOCK

// ---- Tests/Collections/ByteListClearTest.TcPOU
(*
SPDX-FileCopyrightText: c 2026 Oleksandr Tiutyk <trofimich@gmail.com>
SPDX-License-Identifier: MIT
License: https://opensource.org/license/mit
*)

(*!
<summary>Checks retained storage reuse and explicit release behavior.</summary>
<description>
Runs against the selected fixture. The base case clears it before publishing the result.
</description>
*)

{attribute 'no_assign'}
{attribute 'no_explicit_call' := 'do not call this function block directly'}
FUNCTION_BLOCK ByteListClearTest EXTENDS ByteListTestCase
VAR_STAT
	{attribute 'hide'}
	_ClassName : STRING := __POUNAME();
END_VAR

(*!
<summary>Checks retained storage reuse and explicit release behavior.</summary>
*)
METHOD PROTECTED ExecuteTest
VAR
	values : ARRAY [0..5] OF BYTE := [0, 1, 2, 3, 4, 5];
	capacity : TOF_Core.DINT_LENGTH;
	buffer : POINTER TO BYTE;
END_VAR
_List.AppendAny(data := values);
capacity := _List.Capacity;
buffer := GetBufferAddress();

Assert.ThatBool(
	actual := capacity >= 6 AND_THEN buffer <> TOF_Core.Memory.NULL_ADDRESS,
	message := "Appending six bytes must provide backing storage"
).IsTrue();

_List.Clear(releaseDynamicMemory := FALSE);

Assert.ThatBool(
	actual := _List.Empty AND_THEN _List.Capacity = capacity AND_THEN GetBufferAddress() = buffer,
	message := "Clear without release must empty the list while retaining storage"
).IsTrue();

_List.AppendByte(value := BYTE#255);

Assert.ThatBool(
	actual := _List.Length = 1
		AND_THEN _List.Get(index := 0) = BYTE#255
		AND_THEN GetBufferAddress() = buffer,
	message := "Appending after a clear must reuse the retained buffer"
).IsTrue();

_List.Clear(releaseDynamicMemory := TRUE);

